C05488=1125.538,-96.139,-46.252,179.561,4.488,148.877
C05489=1125.533,-95.888,-46.261,179.560,4.493,148.878
C05490=1125.527,-95.639,-46.269,179.560,4.499,148.879
C05491=1125.522,-95.389,-46.278,179.560,4.504,148.880
C05492=1125.517,-95.139,-46.287,179.559,4.508,148.882
C05493=1125.511,-94.889,-46.296,179.559,4.513,148.883
C05494=1125.506,-94.639,-46.305,179.559,4.518,148.884
C05495=1125.500,-94.389,-46.314,179.558,4.522,148.885
C05496=1125.495,-94.140,-46.323,179.558,4.528,148.886
C05497=1125.489,-93.890,-46.332,179.557,4.532,148.888
C05498=1125.484,-93.641,-46.341,179.556,4.537,148.889
C05499=1125.478,-93.390,-46.350,179.555,4.542,148.890
C05500=1125.474,-93.141,-46.360,179.555,4.547,148.891
C05501=1125.468,-92.891,-46.369,179.554,4.551,148.893
C05502=1125.463,-92.642,-46.377,179.554,4.556,148.894
C05503=1125.457,-92.392,-46.386,179.552,4.561,148.895
C05504=1125.452,-92.142,-46.395,179.552,4.565,148.896
C05505=1125.446,-91.892,-46.404,179.551,4.570,148.897
C05506=1125.441,-91.642,-46.413,179.551,4.575,148.899
C05507=1125.436,-91.393,-46.422,179.550,4.580,148.900
C05508=1125.431,-91.143,-46.431,179.549,4.585,148.901
C05509=1125.425,-90.893,-46.441,179.548,4.589,148.902
C05510=1125.419,-90.643,-46.449,179.548,4.594,148.904
C05511=1125.414,-90.394,-46.458,179.547,4.599,148.905
C05512=1125.409,-90.144,-46.467,179.547,4.604,148.906
C05513=1125.403,-89.894,-46.477,179.546,4.609,148.907
C05514=1125.398,-89.644,-46.486,179.546,4.614,148.909
C05515=1125.393,-89.394,-46.495,179.544,4.618,148.910
C05516=1125.389,-89.179,-46.503,179.544,4.622,148.911
C05517=1125.383,-88.963,-46.511,179.543,4.627,148.912
C05518=1125.379,-88.747,-46.518,179.544,4.632,148.913
C05519=1125.374,-88.532,-46.526,179.543,4.636,148.914
C05520=1125.370,-88.316,-46.534,179.543,4.640,148.915
C05521=1125.365,-88.100,-46.542,179.542,4.644,148.916
C05522=1125.360,-87.885,-46.550,179.542,4.648,148.917
C05523=1125.356,-87.669,-46.558,179.541,4.653,148.919
C05524=1125.350,-87.419,-46.567,179.541,4.658,148.920
C05525=1125.345,-87.169,-46.576,179.540,4.662,148.921
C05526=1125.339,-86.919,-46.585,179.540,4.667,148.922
C05527=1125.335,-86.670,-46.595,179.539,4.672,148.923
C05528=1125.329,-86.420,-46.604,179.538,4.677,148.925
C05529=1125.323,-86.170,-46.613,179.538,4.682,148.926
C05530=1125.318,-85.920,-46.622,179.538,4.687,148.927
C05531=1125.313,-85.670,-46.631,179.538,4.693,148.928
C05532=1125.308,-85.421,-46.641,179.537,4.697,148.929
C05533=1125.302,-85.171,-46.650,179.537,4.702,148.931
C05534=1125.297,-84.922,-46.659,179.536,4.707,148.932
C05535=1125.291,-84.671,-46.668,179.536,4.713,148.933
C05536=1125.286,-84.422,-46.678,179.535,4.717,148.934
C05537=1125.281,-84.172,-46.687,179.535,4.722,148.935
C05538=1125.275,-83.922,-46.696,179.535,4.728,148.937
C05539=1125.270,-83.673,-46.706,179.535,4.733,148.938
C05540=1125.264,-83.423,-46.715,179.534,4.738,148.939
C05541=1125.259,-83.173,-46.724,179.534,4.743,148.940
C05542=1125.254,-82.924,-46.734,179.533,4.747,148.941
C05543=1125.248,-82.674,-46.743,179.533,4.753,148.942
C05544=1125.243,-82.424,-46.752,179.533,4.758,148.944
C05545=1125.237,-82.174,-46.763,179.532,4.763,148.945
C05546=1125.232,-81.924,-46.771,179.532,4.768,148.946
C05547=1125.227,-81.674,-46.780,179.532,4.774,148.947
C05548=1125.221,-81.425,-46.791,179.532,4.779,148.949
C05549=1125.216,-81.175,-46.799,179.532,4.784,148.950
C05550=1125.210,-80.925,-46.809,179.532,4.789,148.951
C05551=1125.205,-80.676,-46.819,179.531,4.794,148.952
C05552=1125.200,-80.425,-46.828,179.531,4.799,148.953
C05553=1125.195,-80.176,-46.838,179.531,4.805,148.954
C05554=1125.190,-79.926,-46.847,179.531,4.810,148.956
C05555=1125.184,-79.676,-46.856,179.531,4.815,148.957
C05556=1125.179,-79.426,-46.866,179.531,4.820,148.958
C05557=1125.173,-79.176,-46.876,179.530,4.825,148.959
C05558=1125.169,-78.927,-46.885,179.530,4.830,148.960
C05559=1125.163,-78.677,-46.895,179.530,4.836,148.961
C05560=1125.158,-78.427,-46.904,179.530,4.841,148.963
C05561=1125.152,-78.177,-46.914,179.530,4.846,148.964
C05562=1125.147,-77.928,-46.923,179.530,4.851,148.965
C05563=1125.141,-77.678,-46.933,179.530,4.856,148.966
C05564=1125.136,-77.429,-46.942,179.530,4.861,148.967
C05565=1125.130,-77.179,-46.952,179.530,4.867,148.968
C05566=1125.125,-76.929,-46.962,179.530,4.872,148.969
C05567=1125.120,-76.679,-46.971,179.530,4.877,148.970
C05568=1125.114,-76.430,-46.981,179.530,4.882,148.972
C05569=1125.109,-76.180,-46.990,179.530,4.888,148.973
C05570=1125.104,-75.930,-47.001,179.530,4.892,148.974
C05571=1125.099,-75.680,-47.010,179.530,4.898,148.975
C05572=1125.093,-75.465,-47.019,179.530,4.902,148.976
C05573=1125.089,-75.249,-47.027,179.530,4.907,148.977
C05574=1125.084,-75.033,-47.035,179.530,4.911,148.978
C05575=1125.080,-74.817,-47.043,179.530,4.916,148.979
C05576=1125.075,-74.602,-47.052,179.531,4.921,148.980
C05577=1125.071,-74.387,-47.060,179.530,4.925,148.981
C05578=1125.066,-74.170,-47.069,179.531,4.930,148.982
C05579=1125.062,-73.955,-47.077,179.531,4.934,148.983
C05580=1125.056,-73.705,-47.087,179.531,4.940,148.984
C05581=1125.050,-73.456,-47.097,179.531,4.945,148.985
C05582=1125.045,-73.206,-47.107,179.532,4.950,148.986
C05583=1125.039,-72.956,-47.116,179.532,4.955,148.987
C05584=1125.035,-72.706,-47.126,179.531,4.961,148.988
C05585=1125.030,-72.457,-47.136,179.532,4.966,148.989
C05586=1125.024,-72.207,-47.146,179.532,4.971,148.990
C05587=1125.019,-71.957,-47.155,179.532,4.976,148.991
C05588=1125.013,-71.708,-47.166,179.533,4.982,148.992
C05589=1125.007,-71.458,-47.175,179.533,4.987,148.993
C05590=1125.002,-71.207,-47.186,179.533,4.992,148.995
C05591=1124.997,-70.958,-47.195,179.534,4.998,148.996
C05592=1124.992,-70.709,-47.205,179.534,5.003,148.997
C05593=1124.986,-70.458,-47.215,179.535,5.009,148.998
C05594=1124.982,-70.208,-47.225,179.534,5.014,148.999
C05595=1124.976,-69.959,-47.235,179.535,5.019,149.000
C05596=1124.971,-69.709,-47.245,179.535,5.025,149.001
C05597=1124.965,-69.460,-47.256,179.536,5.029,149.002
C05598=1124.960,-69.210,-47.264,179.536,5.035,149.003
C05599=1124.955,-68.960,-47.275,179.536,5.040,149.004
C05600=1124.949,-68.710,-47.285,179.537,5.046,149.005
C05601=1124.944,-68.461,-47.295,179.537,5.051,149.006
C05602=1124.939,-68.211,-47.305,179.538,5.057,149.007
C05603=1124.934,-67.961,-47.316,179.538,5.061,149.008
C05604=1124.928,-67.711,-47.325,179.539,5.067,149.009
C05605=1124.922,-67.461,-47.335,179.539,5.072,149.010
C05606=1124.917,-67.212,-47.345,179.540,5.078,149.011
C05607=1124.912,-66.962,-47.356,179.540,5.083,149.012
C05608=1124.907,-66.712,-47.366,179.541,5.089,149.013
C05609=1124.901,-66.463,-47.376,179.541,5.093,149.014
C05610=1124.896,-66.213,-47.387,179.542,5.099,149.015
C05611=1124.891,-65.963,-47.397,179.543,5.104,149.016
C05612=1124.886,-65.714,-47.406,179.543,5.110,149.017
C05613=1124.881,-65.464,-47.417,179.543,5.114,149.018
C05614=1124.875,-65.214,-47.427,179.544,5.120,149.019
C05615=1124.869,-64.965,-47.437,179.545,5.125,149.020
C05616=1124.864,-64.714,-47.448,179.545,5.131,149.021
C05617=1124.859,-64.465,-47.458,179.546,5.136,149.022
C05618=1124.853,-64.215,-47.468,179.547,5.141,149.023
C05619=1124.848,-63.965,-47.479,179.548,5.147,149.024
C05620=1124.843,-63.716,-47.489,179.549,5.152,149.024
C05621=1124.838,-63.466,-47.499,179.549,5.157,149.025
C05622=1124.833,-63.216,-47.509,179.550,5.162,149.026
C05623=1124.827,-62.966,-47.519,179.551,5.168,149.027
C05624=1124.822,-62.717,-47.530,179.551,5.173,149.028
C05625=1124.817,-62.467,-47.540,179.552,5.178,149.029
C05626=1124.811,-62.218,-47.551,179.553,5.184,149.030
C05627=1124.806,-61.967,-47.562,179.554,5.189,149.031
C05628=1124.801,-61.751,-47.570,179.554,5.193,149.032
C05629=1124.797,-61.536,-47.580,179.555,5.198,149.032
C05630=1124.793,-61.321,-47.588,179.556,5.203,149.033
C05631=1124.788,-61.106,-47.597,179.557,5.208,149.034
C05632=1124.783,-60.890,-47.607,179.558,5.212,149.035
C05633=1124.778,-60.675,-47.616,179.559,5.216,149.035
C05634=1124.773,-60.459,-47.624,179.559,5.221,149.036
C05635=1124.769,-60.244,-47.633,179.560,5.226,149.037
C05636=1124.765,-59.994,-47.644,179.559,5.230,149.038
C05637=1124.759,-59.744,-47.655,179.560,5.235,149.039
C05638=1124.754,-59.494,-47.665,179.559,5.240,149.040
C05639=1124.749,-59.245,-47.675,179.559,5.244,149.041
C05640=1124.743,-58.994,-47.687,179.559,5.249,149.042
C05641=1124.738,-58.745,-47.697,179.558,5.253,149.043
C05642=1124.733,-58.495,-47.708,179.559,5.258,149.044
C05643=1124.727,-58.245,-47.718,179.558,5.262,149.046
C05644=1124.722,-57.996,-47.730,179.558,5.268,149.047
C05645=1124.717,-57.746,-47.740,179.558,5.271,149.048
C05646=1124.712,-57.496,-47.750,179.558,5.277,149.049
C05647=1124.706,-57.246,-47.761,179.557,5.281,149.050
C05648=1124.701,-56.997,-47.772,179.557,5.286,149.051
C05649=1124.696,-56.747,-47.782,179.557,5.291,149.052
C05650=1124.691,-56.497,-47.793,179.557,5.295,149.053
C05651=1124.685,-56.248,-47.804,179.557,5.300,149.054
C05652=1124.680,-55.998,-47.814,179.556,5.304,149.055
C05653=1124.675,-55.748,-47.824,179.556,5.309,149.056
C05654=1124.669,-55.498,-47.836,179.556,5.313,149.057
C05655=1124.664,-55.249,-47.846,179.556,5.319,149.058
C05656=1124.659,-54.999,-47.857,179.556,5.324,149.060
C05657=1124.654,-54.750,-47.868,179.556,5.328,149.060
C05658=1124.649,-54.499,-47.879,179.556,5.333,149.062
C05659=1124.643,-54.250,-47.889,179.555,5.337,149.063
C05660=1124.638,-54.000,-47.900,179.555,5.342,149.064
C05661=1124.632,-53.750,-47.911,179.555,5.346,149.065
C05662=1124.627,-53.501,-47.922,179.555,5.351,149.066
C05663=1124.622,-53.251,-47.932,179.554,5.355,149.067
C05664=1124.617,-53.002,-47.944,179.554,5.361,149.068
C05665=1124.611,-52.752,-47.954,179.554,5.366,149.069
C05666=1124.607,-52.502,-47.965,179.554,5.370,149.070
C05667=1124.600,-52.253,-47.976,179.554,5.375,149.071
C05668=1124.595,-52.002,-47.986,179.553,5.379,149.072
C05669=1124.590,-51.753,-47.997,179.553,5.384,149.074
C05670=1124.585,-51.503,-48.008,179.553,5.388,149.074
C05671=1124.580,-51.254,-48.019,179.553,5.393,149.076
C05672=1124.574,-51.004,-48.030,179.553,5.398,149.077
C05673=1124.569,-50.754,-48.041,179.553,5.402,149.078
C05674=1124.564,-50.504,-48.052,179.553,5.408,149.079
C05675=1124.559,-50.255,-48.063,179.552,5.412,149.080
C05676=1124.553,-50.005,-48.074,179.552,5.417,149.081
C05677=1124.548,-49.755,-48.085,179.552,5.421,149.082
C05678=1124.543,-49.505,-48.096,179.552,5.426,149.083
C05679=1124.538,-49.256,-48.106,179.551,5.431,149.084
C05680=1124.532,-49.006,-48.118,179.551,5.435,149.085
C05681=1124.527,-48.757,-48.129,179.551,5.440,149.086
C05682=1124.522,-48.507,-48.140,179.551,5.445,149.088
C05683=1124.517,-48.257,-48.150,179.551,5.450,149.088
C05684=1124.512,-48.041,-48.160,179.551,5.453,149.089
C05685=1124.508,-47.827,-48.170,179.550,5.458,149.090
C05686=1124.503,-47.611,-48.179,179.550,5.462,149.091
C05687=1124.498,-47.395,-48.189,179.550,5.466,149.092
C05688=1124.493,-47.180,-48.198,179.550,5.470,149.093
C05689=1124.489,-46.964,-48.207,179.550,5.474,149.094
C05690=1124.484,-46.749,-48.217,179.550,5.478,149.095
C05691=1124.480,-46.534,-48.227,179.550,5.482,149.096
C05692=1124.475,-46.284,-48.238,179.549,5.487,149.097
C05693=1124.470,-46.034,-48.249,179.549,5.491,149.098
C05694=1124.464,-45.785,-48.260,179.549,5.496,149.099
C05695=1124.459,-45.535,-48.271,179.549,5.501,149.100
C05696=1124.454,-45.285,-48.282,179.549,5.506,149.101
C05697=1124.448,-45.036,-48.294,179.548,5.510,149.102
C05698=1124.443,-44.785,-48.304,179.548,5.515,149.103
C05699=1124.439,-44.536,-48.315,179.548,5.519,149.105
C05700=1124.433,-44.287,-48.327,179.548,5.525,149.106
C05701=1124.428,-44.037,-48.338,179.548,5.529,149.107
C05702=1124.423,-43.787,-48.349,179.547,5.534,149.108
C05703=1124.417,-43.537,-48.360,179.547,5.539,149.109
C05704=1124.412,-43.288,-48.372,179.547,5.543,149.110
C05705=1124.406,-43.037,-48.383,179.548,5.549,149.111
C05706=1124.401,-42.788,-48.394,179.549,5.554,149.112
C05707=1124.396,-42.539,-48.405,179.551,5.560,149.112
C05708=1124.391,-42.289,-48.417,179.552,5.565,149.113
C05709=1124.385,-42.039,-48.427,179.555,5.571,149.114
C05710=1124.380,-41.789,-48.439,179.556,5.577,149.115
C05711=1124.375,-41.540,-48.450,179.558,5.583,149.115
C05712=1124.370,-41.290,-48.462,179.559,5.588,149.116
C05713=1124.365,-41.041,-48.473,179.561,5.594,149.117
C05714=1124.359,-40.791,-48.485,179.563,5.599,149.117
C05715=1124.354,-40.541,-48.495,179.564,5.605,149.118
C05716=1124.349,-40.291,-48.507,179.566,5.610,149.119
C05717=1124.343,-40.042,-48.518,179.567,5.615,149.120
C05718=1124.338,-39.792,-48.530,179.568,5.621,149.121
C05719=1124.333,-39.542,-48.541,179.570,5.626,149.121
C05720=1124.328,-39.292,-48.553,179.571,5.631,149.122
C05721=1124.323,-39.043,-48.564,179.572,5.636,149.123
C05722=1124.317,-38.793,-48.576,179.574,5.642,149.123
C05723=1124.312,-38.544,-48.587,179.575,5.647,149.124
C05724=1124.307,-38.294,-48.599,179.576,5.651,149.125
C05725=1124.302,-38.044,-48.611,179.577,5.657,149.126
C05726=1124.296,-37.795,-48.622,179.578,5.661,149.127
C05727=1124.291,-37.545,-48.634,179.579,5.667,149.127
C05728=1124.286,-37.295,-48.645,179.580,5.672,149.128
C05729=1124.281,-37.045,-48.657,179.581,5.676,149.129
C05730=1124.275,-36.796,-48.669,179.582,5.681,149.130
C05731=1124.271,-36.546,-48.680,179.583,5.686,149.130
C05732=1124.265,-36.297,-48.692,179.584,5.691,149.131
C05733=1124.260,-36.047,-48.703,179.585,5.695,149.132
C05734=1124.254,-35.797,-48.715,179.585,5.700,149.133
C05735=1124.249,-35.547,-48.727,179.586,5.706,149.134
C05736=1124.244,-35.298,-48.738,179.587,5.710,149.134
C05737=1124.239,-35.048,-48.750,179.588,5.715,149.135
C05738=1124.234,-34.798,-48.763,179.588,5.720,149.136
C05739=1124.229,-34.549,-48.774,179.589,5.724,149.137
C05740=1124.224,-34.333,-48.785,179.589,5.728,149.138
C05741=1124.219,-34.118,-48.794,179.589,5.731,149.138
C05742=1124.215,-33.903,-48.804,179.590,5.736,149.139
C05743=1124.211,-33.687,-48.815,179.590,5.739,149.140
C05744=1124.206,-33.472,-48.825,179.590,5.743,149.141
C05745=1124.201,-33.257,-48.835,179.591,5.747,149.141
C05746=1124.197,-33.041,-48.845,179.591,5.750,149.142
C05747=1124.193,-32.826,-48.855,179.591,5.755,149.143
C05748=1124.187,-32.576,-48.867,179.591,5.759,149.144
C05749=1124.182,-32.326,-48.879,179.592,5.764,149.145
C05750=1124.177,-32.077,-48.892,179.592,5.768,149.146
C05751=1124.172,-31.827,-48.903,179.592,5.773,149.147
C05752=1124.167,-31.577,-48.915,179.592,5.776,149.147
C05753=1124.161,-31.327,-48.927,179.592,5.780,149.148
C05754=1124.156,-31.078,-48.939,179.592,5.785,149.149
C05755=1124.151,-30.828,-48.950,179.592,5.789,149.150
C05756=1124.145,-30.579,-48.962,179.591,5.793,149.151
C05757=1124.140,-30.329,-48.974,179.591,5.797,149.152
C05758=1124.135,-30.080,-48.986,179.592,5.802,149.153
C05759=1124.130,-29.830,-48.998,179.592,5.806,149.154
C05760=1124.125,-29.580,-49.010,179.591,5.810,149.155
C05761=1124.120,-29.331,-49.022,179.591,5.814,149.156
C05762=1124.114,-29.081,-49.034,179.590,5.819,149.157
C05763=1124.109,-28.831,-49.046,179.590,5.823,149.158
C05764=1124.104,-28.582,-49.057,179.589,5.826,149.159
C05765=1124.099,-28.332,-49.070,179.588,5.831,149.160
C05766=1124.093,-28.082,-49.082,179.588,5.834,149.161
C05767=1124.088,-27.832,-49.094,179.587,5.839,149.162
C05768=1124.083,-27.583,-49.106,179.587,5.843,149.164
C05769=1124.078,-27.333,-49.118,179.586,5.847,149.165
C05770=1124.073,-27.084,-49.129,179.585,5.851,149.166
C05771=1124.068,-26.834,-49.142,179.585,5.855,149.167
C05772=1124.062,-26.584,-49.154,179.584,5.858,149.168
C05773=1124.057,-26.335,-49.167,179.583,5.863,149.169
C05774=1124.052,-26.085,-49.178,179.581,5.867,149.170
C05775=1124.047,-25.835,-49.190,179.582,5.871,149.171
C05776=1124.042,-25.586,-49.202,179.582,5.876,149.172
C05777=1124.036,-25.336,-49.214,179.583,5.881,149.173
C05778=1124.031,-25.086,-49.226,179.584,5.886,149.174
C05779=1124.026,-24.837,-49.239,179.584,5.891,149.175
C05780=1124.020,-24.587,-49.251,179.585,5.896,149.175
C05781=1124.015,-24.338,-49.263,179.586,5.901,149.176
C05782=1124.010,-24.088,-49.275,179.587,5.906,149.177
C05783=1124.006,-23.839,-49.287,179.587,5.911,149.178
C05784=1124.000,-23.589,-49.299,179.588,5.915,149.179
C05785=1123.995,-23.339,-49.312,179.589,5.921,149.180
C05786=1123.990,-23.090,-49.323,179.590,5.925,149.181
C05787=1123.984,-22.840,-49.336,179.590,5.930,149.182
C05788=1123.979,-22.590,-49.348,179.591,5.935,149.182
C05789=1123.974,-22.341,-49.361,179.592,5.940,149.183
C05790=1123.969,-22.090,-49.373,179.592,5.945,149.184
C05791=1123.964,-21.841,-49.385,179.593,5.950,149.185
C05792=1123.958,-21.591,-49.397,179.594,5.954,149.186
C05793=1123.953,-21.342,-49.410,179.595,5.960,149.187
C05794=1123.948,-21.092,-49.422,179.595,5.964,149.188
C05795=1123.943,-20.842,-49.434,179.596,5.969,149.188
C05796=1123.938,-20.627,-49.445,179.597,5.973,149.189
C05797=1123.934,-20.412,-49.455,179.597,5.977,149.190
C05798=1123.929,-20.197,-49.466,179.598,5.981,149.190
C05799=1123.925,-19.982,-49.477,179.598,5.985,149.191
C05800=1123.920,-19.766,-49.488,179.599,5.990,149.192
C05801=1123.916,-19.551,-49.499,179.600,5.994,149.193
C05802=1123.912,-19.336,-49.509,179.600,5.997,149.193
C05803=1123.907,-19.120,-49.520,179.601,6.002,149.194
C05804=1123.902,-18.870,-49.532,179.602,6.007,149.195
C05805=1123.897,-18.621,-49.545,179.602,6.011,149.196
C05806=1123.891,-18.371,-49.557,179.603,6.016,149.197
C05807=1123.886,-18.122,-49.569,179.603,6.021,149.198
C05808=1123.881,-17.873,-49.582,179.605,6.026,149.198
C05809=1123.876,-17.623,-49.594,179.605,6.031,149.199
C05810=1123.870,-17.372,-49.607,179.606,6.035,149.200
C05811=1123.865,-17.123,-49.620,179.607,6.040,149.201
C05812=1123.860,-16.874,-49.633,179.607,6.044,149.202
C05813=1123.855,-16.624,-49.644,179.608,6.049,149.202
C05814=1123.850,-16.374,-49.657,179.608,6.054,149.203
C05815=1123.845,-16.125,-49.670,179.609,6.058,149.204
C05816=1123.840,-15.875,-49.683,179.610,6.064,149.205
C05817=1123.835,-15.625,-49.694,179.611,6.069,149.206
C05818=1123.829,-15.376,-49.707,179.612,6.073,149.206
C05819=1123.824,-15.126,-49.720,179.612,6.078,149.207
C05820=1123.818,-14.877,-49.733,179.613,6.082,149.208
C05821=1123.814,-14.627,-49.746,179.614,6.087,149.209
C05822=1123.809,-14.378,-49.758,179.614,6.091,149.210
C05823=1123.803,-14.128,-49.770,179.615,6.096,149.211
C05824=1123.798,-13.878,-49.783,179.615,6.101,149.212
C05825=1123.793,-13.628,-49.796,179.616,6.105,149.212
C05826=1123.788,-13.379,-49.809,179.617,6.110,149.213
C05827=1123.783,-13.129,-49.822,179.617,6.115,149.214
C05828=1123.778,-12.880,-49.834,179.618,6.119,149.215
C05829=1123.773,-12.630,-49.847,179.619,6.124,149.216
C05830=1123.767,-12.380,-49.860,179.619,6.128,149.216
C05831=1123.762,-12.131,-49.873,179.620,6.133,149.217
C05832=1123.757,-11.882,-49.886,179.621,6.138,149.218
C05833=1123.752,-11.631,-49.898,179.621,6.142,149.219
C05834=1123.746,-11.381,-49.911,179.622,6.147,149.220
C05835=1123.741,-11.132,-49.924,179.623,6.151,149.220
C05836=1123.737,-10.882,-49.937,179.623,6.156,149.221
C05837=1123.732,-10.633,-49.949,179.624,6.160,149.222
C05838=1123.726,-10.383,-49.962,179.625,6.165,149.223
C05839=1123.721,-10.134,-49.975,179.625,6.170,149.224
C05840=1123.716,-9.884,-49.988,179.626,6.174,149.224
C05841=1123.710,-9.634,-50.001,179.627,6.179,149.225
C05842=1123.705,-9.385,-50.014,179.627,6.184,149.226
C05843=1123.701,-9.135,-50.027,179.628,6.188,149.227
C05844=1123.695,-8.886,-50.041,179.629,6.193,149.228
C05845=1123.690,-8.637,-50.053,179.629,6.197,149.229
C05846=1123.685,-8.387,-50.066,179.630,6.202,149.229
C05847=1123.679,-8.137,-50.079,179.631,6.207,149.230
C05848=1123.674,-7.888,-50.092,179.631,6.211,149.231
C05849=1123.670,-7.638,-50.105,179.632,6.216,149.232
C05850=1123.664,-7.388,-50.118,179.633,6.220,149.233
C05851=1123.659,-7.139,-50.131,179.633,6.225,149.233
C05852=1123.655,-6.923,-50.142,179.634,6.229,149.234
C05853=1123.651,-6.708,-50.154,179.635,6.233,149.235
C05854=1123.645,-6.493,-50.165,179.635,6.236,149.235
C05855=1123.641,-6.278,-50.176,179.636,6.241,149.236
C05856=1123.637,-6.062,-50.188,179.636,6.245,149.237
C05857=1123.632,-5.847,-50.199,179.636,6.248,149.238
C05858=1123.628,-5.632,-50.210,179.637,6.253,149.238
C05859=1123.624,-5.417,-50.221,179.638,6.256,149.239
C05860=1123.619,-5.167,-50.235,179.638,6.261,149.240
C05861=1123.613,-4.918,-50.247,179.639,6.265,149.241
C05862=1123.608,-4.668,-50.261,179.640,6.270,149.241
C05863=1123.603,-4.419,-50.274,179.640,6.275,149.242
C05864=1123.598,-4.169,-50.288,179.641,6.279,149.243
C05865=1123.593,-3.919,-50.300,179.641,6.283,149.244
C05866=1123.587,-3.670,-50.314,179.642,6.288,149.245
C05867=1123.583,-3.420,-50.327,179.642,6.292,149.246
C05868=1123.577,-3.171,-50.340,179.643,6.297,149.246
C05869=1123.572,-2.921,-50.353,179.644,6.301,149.247
C05870=1123.567,-2.671,-50.367,179.644,6.306,149.248
C05871=1123.562,-2.422,-50.380,179.645,6.311,149.249
C05872=1123.557,-2.172,-50.393,179.646,6.315,149.250
C05873=1123.551,-1.923,-50.406,179.646,6.320,149.250
C05874=1123.546,-1.673,-50.420,179.646,6.324,149.251
C05875=1123.541,-1.424,-50.433,179.647,6.328,149.252
C05876=1123.536,-1.173,-50.446,179.648,6.333,149.253
C05877=1123.531,-0.925,-50.460,179.648,6.338,149.254
C05878=1123.526,-0.674,-50.473,179.649,6.342,149.255
C05879=1123.521,-0.425,-50.486,179.650,6.347,149.255
C05880=1123.516,-0.175,-50.500,179.650,6.351,149.256
C05881=1123.511,0.074,-50.513,179.650,6.355,149.257
C05882=1123.506,0.324,-50.527,179.651,6.360,149.258
C05883=1123.500,0.573,-50.540,179.652,6.364,149.259
C05884=1123.495,0.823,-50.553,179.652,6.369,149.260
C05885=1123.490,1.072,-50.567,179.653,6.374,149.260
C05886=1123.485,1.322,-50.580,179.653,6.379,149.261
C05887=1123.480,1.571,-50.594,179.654,6.382,149.262
C05888=1123.475,1.821,-50.607,179.654,6.387,149.263
C05889=1123.470,2.070,-50.621,179.655,6.392,149.264
C05890=1123.464,2.321,-50.635,179.655,6.396,149.265
C05891=1123.460,2.569,-50.648,179.656,6.401,149.265
C05892=1123.454,2.820,-50.661,179.657,6.405,149.266
C05893=1123.449,3.069,-50.675,179.657,6.409,149.267
C05894=1123.444,3.319,-50.688,179.657,6.414,149.268
C05895=1123.439,3.568,-50.702,179.658,6.419,149.269
C05896=1123.434,3.818,-50.716,179.658,6.423,149.270
C05897=1123.429,4.068,-50.729,179.659,6.428,149.270
C05898=1123.423,4.317,-50.743,179.660,6.432,149.271
C05899=1123.418,4.567,-50.757,179.660,6.436,149.272
C05900=1123.413,4.816,-50.769,179.660,6.441,149.273
C05901=1123.408,5.066,-50.784,179.661,6.446,149.274
C05902=1123.403,5.315,-50.798,179.661,6.451,149.275
C05903=1123.398,5.565,-50.811,179.662,6.455,149.275
C05904=1123.393,5.815,-50.825,179.662,6.459,149.276
C05905=1123.388,6.064,-50.838,179.663,6.464,149.277
C05906=1123.383,6.314,-50.852,179.664,6.468,149.278
C05907=1123.378,6.563,-50.866,179.664,6.473,149.279
C05908=1123.374,6.778,-50.877,179.664,6.477,149.280
C05909=1123.369,6.994,-50.890,179.664,6.480,149.280
C05910=1123.364,7.209,-50.901,179.665,6.485,149.281
C05911=1123.360,7.423,-50.913,179.666,6.488,149.282
C05912=1123.356,7.639,-50.924,179.666,6.492,149.283
C05913=1123.351,7.854,-50.937,179.666,6.496,149.283
C05914=1123.347,8.069,-50.949,179.667,6.501,149.284
C05915=1123.343,8.284,-50.961,179.667,6.504,149.285
C05916=1123.337,8.533,-50.975,179.668,6.509,149.286
C05917=1123.332,8.783,-50.988,179.669,6.513,149.286
C05918=1123.328,9.033,-51.002,179.669,6.518,149.287
C05919=1123.322,9.282,-51.016,179.670,6.523,149.288
C05920=1123.317,9.532,-51.030,179.671,6.528,149.289
C05921=1123.312,9.782,-51.044,179.672,6.532,149.290
C05922=1123.306,10.031,-51.058,179.673,6.537,149.291
C05923=1123.302,10.280,-51.071,179.674,6.541,149.291
C05924=1123.297,10.530,-51.085,179.674,6.546,149.292
C05925=1123.292,10.779,-51.099,179.675,6.551,149.293
C05926=1123.286,11.029,-51.113,179.676,6.555,149.294
C05927=1123.281,11.279,-51.127,179.676,6.560,149.295
C05928=1123.276,11.528,-51.141,179.678,6.565,149.295
C05929=1123.271,11.778,-51.155,179.678,6.570,149.296
C05930=1123.267,12.027,-51.169,179.679,6.574,149.297
C05931=1123.261,12.277,-51.182,179.680,6.579,149.298
C05932=1123.256,12.527,-51.197,179.681,6.583,149.298
C05933=1123.251,12.776,-51.211,179.682,6.588,149.299
C05934=1123.246,13.026,-51.225,179.682,6.592,149.300
C05935=1123.240,13.275,-51.239,179.683,6.597,149.301
C05936=1123.235,13.525,-51.253,179.684,6.602,149.302
C05937=1123.230,13.774,-51.268,179.685,6.606,149.302
C05938=1123.225,14.023,-51.282,179.686,6.611,149.303
C05939=1123.220,14.273,-51.296,179.687,6.616,149.304
C05940=1123.215,14.523,-51.310,179.687,6.620,149.305
C05941=1123.210,14.773,-51.324,179.689,6.625,149.305
C05942=1123.204,15.022,-51.338,179.689,6.629,149.306
C05943=1123.199,15.271,-51.353,179.690,6.634,149.307
C05944=1123.195,15.521,-51.367,179.691,6.638,149.308
C05945=1123.190,15.771,-51.381,179.692,6.643,149.308
C05946=1123.185,16.020,-51.395,179.692,6.647,149.309
C05947=1123.179,16.269,-51.409,179.693,6.652,149.310
C05948=1123.174,16.519,-51.424,179.694,6.657,149.311
C05949=1123.169,16.769,-51.438,179.695,6.661,149.311
C05950=1123.164,17.019,-51.452,179.697,6.666,149.312
C05951=1123.159,17.268,-51.466,179.697,6.671,149.313
C05952=1123.154,17.517,-51.480,179.698,6.675,149.314
C05953=1123.149,17.767,-51.495,179.699,6.680,149.314
C05954=1123.144,18.017,-51.509,179.700,6.684,149.315
C05955=1123.139,18.266,-51.523,179.701,6.688,149.316
C05956=1123.134,18.516,-51.537,179.701,6.693,149.317
C05957=1123.128,18.765,-51.551,179.702,6.697,149.317
C05958=1123.124,19.014,-51.566,179.703,6.702,149.318
C05959=1123.119,19.264,-51.581,179.704,6.706,149.319
C05960=1123.114,19.514,-51.595,179.705,6.711,149.319
C05961=1123.109,19.763,-51.609,179.706,6.715,149.320
C05962=1123.104,20.013,-51.623,179.707,6.720,149.321
C05963=1123.098,20.262,-51.638,179.708,6.724,149.322
C05964=1123.094,20.477,-51.650,179.709,6.728,149.322
C05965=1123.089,20.692,-51.663,179.709,6.732,149.323
C05966=1123.085,20.907,-51.675,179.710,6.736,149.324
C05967=1123.080,21.122,-51.688,179.711,6.739,149.324
C05968=1123.076,21.337,-51.700,179.712,6.744,149.325
C05969=1123.072,21.552,-51.713,179.713,6.747,149.325
C05970=1123.068,21.767,-51.725,179.714,6.752,149.326
C05971=1123.063,21.982,-51.738,179.714,6.755,149.327
C05972=1123.058,22.232,-51.752,179.715,6.759,149.327
C05973=1123.053,22.481,-51.767,179.716,6.764,149.328
C05974=1123.048,22.730,-51.782,179.717,6.768,149.329
C05975=1123.043,22.981,-51.796,179.718,6.773,149.329
C05976=1123.038,23.230,-51.811,179.719,6.777,149.330
C05977=1123.033,23.479,-51.826,179.720,6.781,149.331
C05978=1123.028,23.729,-51.840,179.721,6.786,149.331
C05979=1123.023,23.979,-51.854,179.722,6.790,149.332
C05980=1123.018,24.228,-51.870,179.723,6.795,149.333
C05981=1123.013,24.478,-51.884,179.724,6.799,149.334
C05982=1123.008,24.728,-51.898,179.725,6.804,149.334
C05983=1123.003,24.976,-51.913,179.726,6.808,149.335
C05984=1122.997,25.226,-51.928,179.727,6.813,149.336
C05985=1122.992,25.475,-51.943,179.728,6.818,149.336
C05986=1122.987,25.725,-51.957,179.729,6.822,149.337
C05987=1122.982,25.974,-51.971,179.730,6.826,149.338
C05988=1122.977,26.224,-51.987,179.731,6.830,149.338
C05989=1122.972,26.474,-52.001,179.732,6.835,149.339
C05990=1122.967,26.723,-52.016,179.733,6.839,149.340
C05991=1122.962,26.973,-52.031,179.734,6.843,149.340
C05992=1122.957,27.222,-52.046,179.735,6.848,149.341
C05993=1122.952,27.471,-52.060,179.736,6.852,149.342
C05994=1122.947,27.721,-52.076,179.737,6.857,149.342
C05995=1122.942,27.971,-52.090,179.738,6.861,149.343
C05996=1122.937,28.220,-52.105,179.739,6.865,149.344
C05997=1122.932,28.470,-52.120,179.740,6.870,149.344
C05998=1122.927,28.719,-52.135,179.741,6.874,149.345
C05999=1122.922,28.969,-52.149,179.742,6.878,149.346
C06000=1122.917,29.218,-52.165,179.743,6.883,149.346
C06001=1122.912,29.468,-52.179,179.744,6.887,149.347
C06002=1122.906,29.717,-52.195,179.745,6.891,149.348
C06003=1122.902,29.966,-52.210,179.746,6.896,149.348
C06004=1122.897,30.217,-52.225,179.748,6.900,149.349
C06005=1122.892,30.466,-52.240,179.749,6.904,149.350
C06006=1122.887,30.716,-52.254,179.750,6.909,149.350
C06007=1122.881,30.965,-52.270,179.751,6.913,149.351
C06008=1122.877,31.214,-52.285,179.752,6.917,149.352
C06009=1122.871,31.464,-52.300,179.753,6.921,149.352
C06010=1122.866,31.713,-52.315,179.754,6.926,149.353
C06011=1122.862,31.962,-52.330,179.755,6.930,149.354
C06012=1122.856,32.212,-52.345,179.756,6.934,149.354
C06013=1122.851,32.461,-52.360,179.757,6.939,149.355
C06014=1122.846,32.711,-52.375,179.758,6.943,149.355
C06015=1122.841,32.961,-52.390,179.759,6.947,149.356
C06016=1122.836,33.211,-52.406,179.760,6.951,149.357
C06017=1122.832,33.460,-52.421,179.761,6.955,149.357
C06018=1122.826,33.709,-52.436,179.762,6.959,149.358
C06019=1122.821,33.959,-52.450,179.763,6.964,149.359
C06020=1122.817,34.173,-52.464,179.764,6.968,149.359
C06021=1122.812,34.388,-52.477,179.765,6.971,149.360
C06022=1122.808,34.603,-52.490,179.766,6.975,149.360
C06023=1122.804,34.819,-52.503,179.767,6.979,149.361
C06024=1122.799,35.034,-52.516,179.768,6.983,149.361
C06025=1122.796,35.248,-52.530,179.769,6.986,149.362
C06026=1122.791,35.463,-52.543,179.770,6.989,149.362
C06027=1122.786,35.678,-52.556,179.771,6.993,149.363
C06028=1122.781,35.927,-52.571,179.772,6.997,149.363
C06029=1122.777,36.177,-52.587,179.773,7.002,149.364
C06030=1122.772,36.426,-52.602,179.774,7.006,149.365
C06031=1122.766,36.676,-52.617,179.775,7.010,149.365
C06032=1122.761,36.925,-52.632,179.777,7.015,149.366
C06033=1122.756,37.175,-52.648,179.778,7.019,149.367
C06034=1122.751,37.424,-52.663,179.779,7.023,149.367
C06035=1122.746,37.674,-52.678,179.780,7.027,149.368
C06036=1122.741,37.923,-52.694,179.781,7.031,149.368
C06037=1122.736,38.172,-52.709,179.782,7.035,149.369
C06038=1122.731,38.422,-52.725,179.783,7.039,149.370
C06039=1122.726,38.671,-52.740,179.784,7.044,149.370
C06040=1122.722,38.921,-52.756,179.785,7.048,149.371
C06041=1122.716,39.170,-52.771,179.786,7.052,149.371
C06042=1122.711,39.420,-52.787,179.788,7.056,149.372
C06043=1122.706,39.669,-52.802,179.789,7.061,149.373
C06044=1122.701,39.919,-52.818,179.790,7.064,149.373
C06045=1122.696,40.168,-52.833,179.791,7.069,149.374
C06046=1122.691,40.418,-52.848,179.792,7.073,149.374
C06047=1122.686,40.667,-52.864,179.793,7.077,149.375
C06048=1122.681,40.917,-52.880,179.795,7.081,149.376
C06049=1122.676,41.166,-52.895,179.796,7.086,149.376
C06050=1122.671,41.416,-52.910,179.797,7.090,149.377
C06051=1122.666,41.665,-52.926,179.798,7.094,149.377
C06052=1122.661,41.915,-52.942,179.800,7.098,149.378
C06053=1122.656,42.164,-52.958,179.801,7.102,149.379
C06054=1122.651,42.414,-52.973,179.802,7.107,149.379
C06055=1122.646,42.664,-52.989,179.803,7.111,149.380
C06056=1122.641,42.912,-53.005,179.804,7.115,149.380
C06057=1122.636,43.162,-53.020,179.806,7.119,149.381
C06058=1122.631,43.411,-53.035,179.806,7.123,149.382
C06059=1122.626,43.661,-53.051,179.808,7.127,149.382
C06060=1122.621,43.910,-53.067,179.809,7.131,149.383
C06061=1122.616,44.160,-53.083,179.810,7.135,149.383
C06062=1122.611,44.409,-53.099,179.811,7.139,149.384
C06063=1122.606,44.658,-53.114,179.812,7.144,149.384
C06064=1122.601,44.908,-53.130,179.813,7.148,149.385
C06065=1122.596,45.158,-53.146,179.815,7.152,149.385
C06066=1122.591,45.407,-53.161,179.816,7.156,149.386
C06067=1122.586,45.656,-53.178,179.817,7.160,149.387
C06068=1122.581,45.906,-53.194,179.819,7.164,149.387
C06069=1122.576,46.156,-53.209,179.820,7.169,149.388
C06070=1122.572,46.405,-53.225,179.821,7.173,149.388
C06071=1122.566,46.654,-53.241,179.822,7.177,149.389
C06072=1122.561,46.904,-53.256,179.823,7.181,149.390
C06073=1122.556,47.154,-53.272,179.825,7.185,149.390
C06074=1122.551,47.402,-53.289,179.826,7.189,149.391
C06075=1122.546,47.652,-53.304,179.827,7.193,149.391
C06076=1122.542,47.867,-53.318,179.828,7.197,149.392
C06077=1122.538,48.081,-53.332,179.829,7.200,149.392
C06078=1122.534,48.297,-53.345,179.831,7.204,149.393
C06079=1122.529,48.512,-53.360,179.831,7.207,149.393
C06080=1122.524,48.726,-53.373,179.832,7.210,149.394
C06081=1122.520,48.942,-53.387,179.834,7.214,149.394
C06082=1122.516,49.156,-53.400,179.834,7.218,149.395
C06083=1122.512,49.370,-53.414,179.836,7.222,149.395
C06084=1122.507,49.620,-53.430,179.836,7.225,149.396
C06085=1122.502,49.869,-53.446,179.838,7.229,149.396
C06086=1122.497,50.119,-53.462,179.839,7.233,149.397
C06087=1122.492,50.368,-53.479,179.840,7.237,149.397
C06088=1122.487,50.618,-53.495,179.842,7.241,149.398
C06089=1122.482,50.867,-53.511,179.843,7.246,149.398
C06090=1122.477,51.117,-53.527,179.844,7.250,149.399
C06091=1122.472,51.366,-53.543,179.845,7.254,149.399
C06092=1122.468,51.616,-53.559,179.847,7.258,149.400
C06093=1122.463,51.865,-53.575,179.848,7.262,149.401
C06094=1122.457,52.114,-53.591,179.849,7.266,149.401
C06095=1122.453,52.364,-53.608,179.851,7.270,149.402
C06096=1122.447,52.613,-53.623,179.852,7.275,149.402
C06097=1122.442,52.863,-53.641,179.853,7.279,149.403
C06098=1122.437,53.112,-53.656,179.855,7.283,149.403
C06099=1122.432,53.362,-53.673,179.855,7.286,149.404
C06100=1122.427,53.610,-53.689,179.857,7.290,149.404
C06101=1122.422,53.860,-53.705,179.858,7.294,149.405
C06102=1122.417,54.109,-53.721,179.859,7.298,149.405
C06103=1122.412,54.359,-53.737,179.861,7.302,149.406
C06104=1122.407,54.608,-53.754,179.862,7.307,149.407
C06105=1122.403,54.858,-53.770,179.863,7.311,149.407
C06106=1122.397,55.108,-53.787,179.864,7.315,149.408
C06107=1122.392,55.357,-53.803,179.866,7.319,149.408
C06108=1122.388,55.606,-53.820,179.867,7.323,149.409
C06109=1122.382,55.856,-53.835,179.869,7.327,149.409
C06110=1122.378,56.105,-53.852,179.870,7.331,149.410
C06111=1122.373,56.354,-53.868,179.871,7.335,149.410
C06112=1122.368,56.604,-53.884,179.872,7.340,149.411
C06113=1122.362,56.853,-53.901,179.873,7.343,149.411
C06114=1122.358,57.103,-53.918,179.875,7.347,149.412
C06115=1122.353,57.352,-53.935,179.876,7.351,149.412
C06116=1122.348,57.602,-53.950,179.878,7.355,149.413
C06117=1122.343,57.851,-53.967,179.879,7.359,149.413
C06118=1122.338,58.100,-53.984,179.880,7.363,149.414
C06119=1122.333,58.350,-54.000,179.881,7.367,149.415
C06120=1122.328,58.600,-54.016,179.883,7.371,149.415
C06121=1122.323,58.849,-54.033,179.884,7.375,149.415
C06122=1122.318,59.098,-54.050,179.886,7.379,149.416
C06123=1122.313,59.347,-54.066,179.887,7.383,149.416
C06124=1122.309,59.597,-54.083,179.888,7.388,149.417
C06125=1122.304,59.846,-54.100,179.890,7.392,149.418
C06126=1122.298,60.095,-54.116,179.891,7.395,149.418
C06127=1122.293,60.345,-54.132,179.892,7.399,149.419
C06128=1122.289,60.595,-54.149,179.893,7.403,149.419
C06129=1122.283,60.844,-54.166,179.895,7.407,149.420
C06130=1122.279,61.093,-54.183,179.896,7.411,149.420
C06131=1122.274,61.343,-54.199,179.898,7.415,149.421
C06132=1122.269,61.557,-54.214,179.899,7.419,149.421
C06133=1122.266,61.772,-54.228,179.900,7.422,149.422
C06134=1122.261,61.986,-54.243,179.901,7.425,149.422
C06135=1122.257,62.202,-54.257,179.902,7.429,149.422
C06136=1122.252,62.416,-54.271,179.903,7.433,149.423
C06137=1122.249,62.631,-54.286,179.905,7.436,149.423
C06138=1122.244,62.845,-54.300,179.906,7.440,149.424
C06139=1122.240,63.060,-54.314,179.907,7.443,149.424
C06140=1122.235,63.310,-54.332,179.908,7.447,149.425
C06141=1122.230,63.559,-54.348,179.909,7.451,149.425
C06142=1122.225,63.808,-54.365,179.911,7.455,149.426
C06143=1122.220,64.058,-54.382,179.912,7.459,149.426
C06144=1122.215,64.308,-54.398,179.914,7.463,149.427
C06145=1122.210,64.557,-54.415,179.915,7.467,149.427
C06146=1122.205,64.806,-54.432,179.917,7.471,149.428
C06147=1122.201,65.055,-54.449,179.918,7.475,149.428
C06148=1122.196,65.305,-54.467,179.919,7.479,149.429
C06149=1122.191,65.554,-54.483,179.921,7.483,149.429
C06150=1122.185,65.803,-54.500,179.922,7.487,149.430
C06151=1122.181,66.053,-54.517,179.923,7.490,149.430
C06152=1122.176,66.303,-54.534,179.925,7.494,149.431
C06153=1122.171,66.551,-54.550,179.926,7.498,149.431
C06154=1122.165,66.801,-54.568,179.927,7.502,149.432
C06155=1122.161,67.050,-54.585,179.929,7.506,149.432
C06156=1122.156,67.300,-54.602,179.930,7.511,149.433
C06157=1122.151,67.549,-54.619,179.931,7.515,149.433
C06158=1122.146,67.799,-54.636,179.933,7.518,149.434
C06159=1122.141,68.048,-54.653,179.934,7.523,149.434
C06160=1122.136,68.297,-54.671,179.936,7.527,149.435
C06161=1122.132,68.547,-54.687,179.937,7.531,149.435
C06162=1122.126,68.796,-54.704,179.939,7.534,149.436
C06163=1122.122,69.045,-54.721,179.940,7.539,149.436
C06164=1122.117,69.294,-54.739,179.942,7.543,149.437
C06165=1122.112,69.544,-54.755,179.943,7.547,149.437
C06166=1122.107,69.794,-54.773,179.944,7.551,149.438
C06167=1122.102,70.044,-54.790,179.945,7.554,149.438
C06168=1122.097,70.292,-54.807,179.947,7.558,149.439
C06169=1122.092,70.541,-54.824,179.948,7.562,149.439
C06170=1122.087,70.791,-54.841,179.949,7.566,149.440
C06171=1122.082,71.040,-54.859,179.951,7.570,149.440
C06172=1122.077,71.290,-54.876,179.953,7.574,149.440
C06173=1122.073,71.539,-54.893,179.954,7.578,149.441
C06174=1122.068,71.789,-54.911,179.955,7.582,149.442
C06175=1122.063,72.037,-54.927,179.957,7.586,149.442
C06176=1122.058,72.287,-54.945,179.958,7.590,149.442
C06177=1122.053,72.536,-54.962,179.960,7.594,149.443
C06178=1122.048,72.786,-54.979,179.961,7.598,149.444
C06179=1122.043,73.035,-54.997,179.963,7.602,149.444
C06180=1122.038,73.285,-55.014,179.964,7.606,149.445
C06181=1122.034,73.534,-55.032,179.965,7.610,149.445
C06182=1122.028,73.783,-55.049,179.967,7.614,149.445
C06183=1122.024,74.033,-55.067,179.969,7.618,149.446
C06184=1122.018,74.282,-55.084,179.970,7.622,149.447
C06185=1122.014,74.531,-55.101,179.971,7.626,149.447
C06186=1122.008,74.780,-55.118,179.973,7.630,149.447
C06187=1122.003,75.030,-55.136,179.974,7.633,149.448
C06188=1122.000,75.245,-55.151,179.975,7.637,149.448
C06189=1121.996,75.459,-55.166,179.976,7.640,149.449
C06190=1121.992,75.674,-55.181,179.978,7.644,149.449
C06191=1121.987,75.888,-55.196,179.979,7.647,149.450
C06192=1121.983,76.103,-55.212,179.980,7.651,149.450
C06193=1121.978,76.318,-55.226,179.981,7.654,149.450
C06194=1121.974,76.533,-55.242,179.982,7.657,149.451
C06195=1121.970,76.747,-55.256,179.984,7.661,149.451
C06196=1121.965,76.996,-55.274,179.985,7.664,149.452
C06197=1121.960,77.246,-55.291,179.986,7.669,149.452
C06198=1121.955,77.495,-55.309,179.986,7.672,149.453
C06199=1121.950,77.744,-55.327,179.987,7.675,149.453
C06200=1121.946,77.993,-55.344,179.989,7.679,149.454
C06201=1121.941,78.243,-55.362,179.990,7.683,149.454
C06202=1121.936,78.492,-55.380,179.991,7.687,149.455
C06203=1121.931,78.742,-55.397,179.992,7.690,149.456
C06204=1121.926,78.991,-55.415,179.993,7.694,149.456
C06205=1121.921,79.240,-55.433,179.994,7.697,149.457
C06206=1121.916,79.489,-55.450,179.995,7.702,149.457
C06207=1121.911,79.739,-55.468,179.995,7.705,149.458
C06208=1121.907,79.988,-55.486,179.997,7.709,149.458
C06209=1121.901,80.237,-55.503,179.997,7.713,149.459
C06210=1121.896,80.487,-55.521,179.999,7.716,149.459
C06211=1121.891,80.736,-55.539,-180.000,7.721,149.460
C06212=1121.887,80.985,-55.557,-179.999,7.724,149.460
C06213=1121.881,81.235,-55.574,-179.998,7.728,149.461
C06214=1121.877,81.485,-55.593,-179.997,7.731,149.462
C06215=1121.873,81.734,-55.610,-179.996,7.736,149.462
C06216=1121.868,81.983,-55.628,-179.994,7.739,149.463
C06217=1121.863,82.232,-55.646,-179.993,7.743,149.463
C06218=1121.858,82.482,-55.663,-179.992,7.747,149.464
C06219=1121.853,82.731,-55.681,-179.991,7.750,149.464
C06220=1121.848,82.980,-55.699,-179.990,7.754,149.465
C06221=1121.843,83.229,-55.717,-179.988,7.758,149.465
C06222=1121.838,83.478,-55.735,-179.988,7.762,149.466
C06223=1121.833,83.728,-55.753,-179.986,7.766,149.466
C06224=1121.828,83.977,-55.770,-179.985,7.769,149.467
C06225=1121.823,84.227,-55.788,-179.984,7.773,149.467
C06226=1121.818,84.476,-55.806,-179.983,7.777,149.468
C06227=1121.814,84.726,-55.825,-179.981,7.781,149.468
C06228=1121.809,84.975,-55.843,-179.980,7.784,149.469
C06229=1121.804,85.224,-55.861,-179.979,7.788,149.469
C06230=1121.799,85.473,-55.879,-179.978,7.792,149.470
C06231=1121.794,85.722,-55.897,-179.976,7.796,149.470
C06232=1121.789,85.971,-55.915,-179.975,7.799,149.471
C06233=1121.784,86.221,-55.933,-179.974,7.804,149.471
C06234=1121.780,86.470,-55.951,-179.972,7.808,149.472
C06235=1121.775,86.720,-55.969,-179.971,7.811,149.472
C06236=1121.770,86.969,-55.987,-179.970,7.815,149.473
C06237=1121.765,87.218,-56.005,-179.969,7.819,149.473
C06238=1121.760,87.467,-56.023,-179.967,7.823,149.474
C06239=1121.756,87.716,-56.041,-179.966,7.827,149.474
C06240=1121.751,87.966,-56.059,-179.964,7.831,149.475
C06241=1121.746,88.215,-56.077,-179.963,7.834,149.475
C06242=1121.741,88.465,-56.096,-179.962,7.838,149.476
C06243=1121.736,88.714,-56.114,-179.961,7.842,149.476
C06244=1121.732,88.929,-56.129,-179.959,7.845,149.477
C06245=1121.728,89.143,-56.145,-179.958,7.849,149.477
C06246=1121.724,89.358,-56.161,-179.957,7.852,149.477
C06247=1121.720,89.572,-56.176,-179.956,7.855,149.478
C06248=1121.715,89.787,-56.191,-179.954,7.859,149.478
C06249=1121.710,90.001,-56.208,-179.953,7.862,149.479
C06250=1121.706,90.216,-56.223,-179.952,7.865,149.479
C06251=1121.702,90.430,-56.239,-179.951,7.869,149.480
C06252=1121.698,90.680,-56.258,-179.949,7.873,149.480
C06253=1121.693,90.929,-56.276,-179.947,7.877,149.480
C06254=1121.688,91.178,-56.294,-179.946,7.880,149.481
C06255=1121.683,91.427,-56.312,-179.945,7.884,149.481
C06256=1121.678,91.677,-56.330,-179.943,7.888,149.482
C06257=1121.674,91.926,-56.349,-179.942,7.892,149.482
C06258=1121.669,92.175,-56.367,-179.940,7.896,149.483
C06259=1121.664,92.424,-56.385,-179.939,7.900,149.483
C06260=1121.659,92.674,-56.404,-179.937,7.904,149.484
C06261=1121.654,92.924,-56.422,-179.936,7.908,149.484
C06262=1121.649,93.172,-56.441,-179.934,7.911,149.485
C06263=1121.644,93.421,-56.459,-179.933,7.915,149.485
C06264=1121.639,93.671,-56.478,-179.931,7.919,149.485
C06265=1121.635,93.920,-56.496,-179.929,7.923,149.486
C06266=1121.630,94.169,-56.514,-179.928,7.927,149.486
C06267=1121.625,94.418,-56.532,-179.926,7.931,149.487
C06268=1121.620,94.668,-56.552,-179.925,7.935,149.487
C06269=1121.615,94.917,-56.570,-179.923,7.939,149.488
C06270=1121.610,95.166,-56.588,-179.921,7.943,149.488
C06271=1121.606,95.416,-56.608,-179.920,7.946,149.488
C06272=1121.601,95.665,-56.626,-179.918,7.950,149.489
C06273=1121.596,95.914,-56.644,-179.917,7.954,149.489
C06274=1121.591,96.164,-56.663,-179.914,7.958,149.489
C06275=1121.586,96.413,-56.681,-179.913,7.962,149.490
C06276=1121.581,96.661,-56.700,-179.911,7.966,149.490
C06277=1121.576,96.912,-56.719,-179.910,7.969,149.491
C06278=1121.571,97.161,-56.737,-179.907,7.974,149.491
C06279=1121.567,97.409,-56.755,-179.906,7.978,149.492
C06280=1121.562,97.660,-56.774,-179.904,7.982,149.492
C06281=1121.557,97.908,-56.793,-179.902,7.985,149.492
C06282=1121.552,98.158,-56.812,-179.901,7.989,149.493
C06283=1121.548,98.407,-56.831,-179.899,7.993,149.493
C06284=1121.543,98.656,-56.849,-179.897,7.997,149.494
C06285=1121.538,98.906,-56.868,-179.895,8.001,149.494
C06286=1121.533,99.154,-56.887,-179.894,8.004,149.494
C06287=1121.528,99.404,-56.906,-179.891,8.009,149.495
C06288=1121.524,99.653,-56.925,-179.890,8.013,149.495
C06289=1121.518,99.902,-56.943,-179.888,8.016,149.495
C06290=1121.514,100.152,-56.962,-179.886,8.020,149.496
C06291=1121.508,100.401,-56.981,-179.885,8.024,149.496
C06292=1121.504,100.650,-57.000,-179.883,8.028,149.496
C06293=1121.499,100.899,-57.019,-179.880,8.032,149.497
C06294=1121.494,101.148,-57.037,-179.879,8.036,149.497
C06295=1121.489,101.398,-57.057,-179.877,8.040,149.497
C06296=1121.485,101.647,-57.076,-179.875,8.044,149.498
C06297=1121.480,101.897,-57.095,-179.873,8.047,149.498
C06298=1121.475,102.145,-57.113,-179.871,8.052,149.499
C06299=1121.470,102.395,-57.133,-179.869,8.055,149.499
C06300=1121.467,102.609,-57.149,-179.867,8.059,149.499
C06301=1121.462,102.824,-57.165,-179.866,8.062,149.499
C06302=1121.458,103.038,-57.181,-179.864,8.065,149.500
C06303=1121.453,103.253,-57.198,-179.863,8.069,149.500
C06304=1121.449,103.467,-57.214,-179.861,8.072,149.500
C06305=1121.445,103.681,-57.231,-179.859,8.076,149.500
C06306=1121.442,103.896,-57.247,-179.857,8.078,149.501
C06307=1121.437,104.110,-57.264,-179.856,8.082,149.501
C06308=1121.433,104.359,-57.282,-179.853,8.086,149.501
C06309=1121.427,104.609,-57.301,-179.851,8.090,149.502
C06310=1121.422,104.858,-57.321,-179.849,8.094,149.502
C06311=1121.418,105.107,-57.340,-179.847,8.097,149.502
C06312=1121.413,105.356,-57.359,-179.845,8.102,149.503
C06313=1121.409,105.605,-57.378,-179.843,8.106,149.503
C06314=1121.403,105.854,-57.397,-179.841,8.109,149.503
C06315=1121.399,106.104,-57.417,-179.839,8.113,149.504
C06316=1121.394,106.354,-57.435,-179.836,8.117,149.504
C06317=1121.389,106.602,-57.455,-179.834,8.121,149.504
C06318=1121.384,106.852,-57.474,-179.832,8.124,149.504
C06319=1121.379,107.101,-57.494,-179.830,8.129,149.505
C06320=1121.375,107.350,-57.513,-179.828,8.132,149.505
C06321=1121.370,107.599,-57.532,-179.826,8.136,149.505
C06322=1121.365,107.849,-57.552,-179.823,8.140,149.505
C06323=1121.361,108.098,-57.571,-179.821,8.144,149.506
C06324=1121.355,108.347,-57.590,-179.819,8.148,149.506
C06325=1121.351,108.596,-57.610,-179.817,8.152,149.506
C06326=1121.345,108.845,-57.629,-179.815,8.155,149.506
C06327=1121.341,109.094,-57.648,-179.812,8.160,149.507
C06328=1121.337,109.344,-57.668,-179.810,8.163,149.507
C06329=1121.331,109.593,-57.687,-179.808,8.167,149.507
C06330=1121.327,109.842,-57.707,-179.805,8.171,149.507
C06331=1121.322,110.091,-57.727,-179.803,8.174,149.508
C06332=1121.318,110.340,-57.746,-179.801,8.179,149.508
C06333=1121.313,110.590,-57.765,-179.799,8.182,149.508
C06334=1121.307,110.838,-57.785,-179.797,8.186,149.508
C06335=1121.303,111.088,-57.804,-179.794,8.190,149.508
C06336=1121.298,111.338,-57.824,-179.792,8.193,149.509
C06337=1121.293,111.586,-57.843,-179.791,8.197,149.509
C06338=1121.288,111.835,-57.864,-179.789,8.200,149.509
C06339=1121.284,112.085,-57.883,-179.787,8.204,149.510
C06340=1121.279,112.333,-57.902,-179.785,8.207,149.510
C06341=1121.274,112.583,-57.922,-179.783,8.211,149.510
C06342=1121.270,112.832,-57.942,-179.781,8.214,149.510
C06343=1121.265,113.082,-57.962,-179.779,8.218,149.511
C06344=1121.260,113.330,-57.981,-179.777,8.222,149.511
C06345=1121.255,113.580,-58.001,-179.776,8.225,149.511
C06346=1121.250,113.829,-58.021,-179.774,8.228,149.511
C06347=1121.245,114.078,-58.040,-179.772,8.232,149.512
C06348=1121.240,114.327,-58.060,-179.770,8.235,149.512
C06349=1121.236,114.576,-58.080,-179.768,8.239,149.512
C06350=1121.231,114.826,-58.100,-179.766,8.242,149.513
C06351=1121.226,115.075,-58.119,-179.764,8.246,149.513
C06352=1121.221,115.324,-58.140,-179.763,8.249,149.513
C06353=1121.217,115.573,-58.159,-179.761,8.253,149.513
C06354=1121.212,115.823,-58.179,-179.759,8.256,149.514
C06355=1121.207,116.071,-58.199,-179.757,8.260,149.514
C06356=1121.203,116.286,-58.216,-179.755,8.262,149.514
C06357=1121.199,116.500,-58.233,-179.754,8.265,149.514
C06358=1121.195,116.714,-58.249,-179.752,8.268,149.515
C06359=1121.191,116.929,-58.267,-179.750,8.271,149.515
C06360=1121.187,117.143,-58.284,-179.749,8.274,149.515
C06361=1121.183,117.357,-58.302,-179.748,8.277,149.515
C06362=1121.178,117.572,-58.318,-179.746,8.280,149.516
C06363=1121.174,117.786,-58.336,-179.744,8.283,149.516
C06364=1121.169,118.035,-58.355,-179.742,8.287,149.516
C06365=1121.165,118.284,-58.376,-179.740,8.290,149.516
C06366=1121.160,118.534,-58.395,-179.739,8.293,149.517
C06367=1121.156,118.783,-58.416,-179.737,8.297,149.517
C06368=1121.150,119.032,-58.435,-179.735,8.300,149.517
C06369=1121.146,119.281,-58.456,-179.733,8.304,149.517
C06370=1121.141,119.530,-58.475,-179.732,8.306,149.518
C06371=1121.136,119.779,-58.496,-179.730,8.310,149.518
C06372=1121.131,120.029,-58.516,-179.728,8.314,149.518
C06373=1121.127,120.278,-58.536,-179.726,8.317,149.519
C06374=1121.122,120.527,-58.556,-179.724,8.321,149.519
C06375=1121.117,120.776,-58.576,-179.722,8.324,149.519
C06376=1121.113,121.025,-58.596,-179.721,8.327,149.519
C06377=1121.108,121.274,-58.616,-179.719,8.331,149.520
C06378=1121.103,121.523,-58.637,-179.717,8.334,149.520
C06379=1121.098,121.772,-58.657,-179.715,8.337,149.520
C06380=1121.094,122.022,-58.677,-179.713,8.341,149.520
C06381=1121.089,122.271,-58.697,-179.712,8.345,149.521
C06382=1121.085,122.520,-58.718,-179.710,8.347,149.521
C06383=1121.079,122.769,-58.737,-179.708,8.351,149.521
C06384=1121.074,123.018,-58.758,-179.706,8.354,149.521
C06385=1121.070,123.267,-58.778,-179.704,8.358,149.522
C06386=1121.065,123.517,-58.798,-179.703,8.361,149.522
C06387=1121.061,123.765,-58.818,-179.701,8.364,149.522
C06388=1121.055,124.015,-58.839,-179.699,8.368,149.523
C06389=1121.051,124.264,-58.860,-179.697,8.371,149.523
C06390=1121.046,124.513,-58.879,-179.696,8.374,149.523
C06391=1121.042,124.762,-58.900,-179.694,8.378,149.523
C06392=1121.037,125.011,-58.921,-179.692,8.381,149.524
C06393=1121.032,125.260,-58.941,-179.690,8.384,149.524
C06394=1121.028,125.509,-58.961,-179.689,8.388,149.524
C06395=1121.023,125.759,-58.981,-179.686,8.392,149.525
C06396=1121.018,126.008,-59.002,-179.685,8.394,149.525
C06397=1121.013,126.257,-59.022,-179.683,8.398,149.525
C06398=1121.009,126.506,-59.043,-179.681,8.402,149.525
C06399=1121.004,126.755,-59.064,-179.680,8.404,149.526
C06400=1120.999,127.004,-59.084,-179.678,8.408,149.526
C06401=1120.995,127.253,-59.104,-179.676,8.411,149.526
C06402=1120.990,127.503,-59.125,-179.675,8.414,149.527
C06403=1120.985,127.752,-59.145,-179.673,8.418,149.527
C06404=1120.981,128.001,-59.165,-179.671,8.421,149.527
C06405=1120.975,128.250,-59.186,-179.669,8.424,149.527
C06406=1120.971,128.499,-59.207,-179.668,8.428,149.528
C06407=1120.966,128.749,-59.228,-179.665,8.431,149.528
C06408=1120.961,128.997,-59.248,-179.664,8.434,149.528
C06409=1120.957,129.246,-59.268,-179.662,8.438,149.528
C06410=1120.952,129.496,-59.289,-179.660,8.442,149.529
C06411=1120.947,129.745,-59.310,-179.659,8.444,149.529
C06412=1120.943,129.958,-59.327,-179.657,8.447,149.529
C06413=1120.939,130.173,-59.346,-179.655,8.450,149.529
C06414=1120.934,130.387,-59.363,-179.654,8.453,149.530
C06415=1120.931,130.601,-59.381,-179.652,8.456,149.530
C06416=1120.926,130.815,-59.398,-179.651,8.459,149.530
C06417=1120.922,131.030,-59.417,-179.650,8.461,149.530
C06418=1120.918,131.245,-59.434,-179.649,8.464,149.531
C06419=1120.914,131.458,-59.452,-179.647,8.467,149.531
C06420=1120.909,131.707,-59.473,-179.645,8.471,149.531
C06421=1120.905,131.956,-59.494,-179.643,8.474,149.531
C06422=1120.900,132.205,-59.515,-179.642,8.477,149.532
C06423=1120.896,132.455,-59.535,-179.640,8.481,149.532
C06424=1120.891,132.704,-59.556,-179.638,8.484,149.532
C06425=1120.886,132.953,-59.577,-179.636,8.487,149.533
C06426=1120.881,133.202,-59.598,-179.635,8.491,149.533
C06427=1120.877,133.451,-59.618,-179.633,8.494,149.533
C06428=1120.872,133.700,-59.640,-179.631,8.497,149.533
C06429=1120.867,133.949,-59.660,-179.630,8.501,149.534
C06430=1120.862,134.198,-59.681,-179.628,8.504,149.534
C06431=1120.858,134.447,-59.702,-179.626,8.507,149.534
C06432=1120.853,134.696,-59.723,-179.625,8.510,149.535
C06433=1120.849,134.945,-59.744,-179.623,8.514,149.535
C06434=1120.844,135.195,-59.765,-179.621,8.518,149.535
C06435=1120.839,135.444,-59.786,-179.620,8.520,149.536
C06436=1120.834,135.693,-59.806,-179.618,8.524,149.536
C06437=1120.829,135.941,-59.828,-179.617,8.527,149.536
C06438=1120.825,136.190,-59.848,-179.615,8.530,149.537
C06439=1120.820,136.440,-59.869,-179.613,8.534,149.537
C06440=1120.815,136.689,-59.891,-179.612,8.537,149.537
C06441=1120.811,136.938,-59.912,-179.610,8.540,149.537
C06442=1120.806,137.187,-59.933,-179.609,8.544,149.538
C06443=1120.801,137.436,-59.953,-179.607,8.547,149.538
C06444=1120.797,137.685,-59.975,-179.605,8.550,149.538
C06445=1120.792,137.935,-59.996,-179.603,8.554,149.539
C06446=1120.788,138.183,-60.017,-179.601,8.557,149.539
C06447=1120.783,138.432,-60.038,-179.600,8.560,149.539
C06448=1120.777,138.682,-60.059,-179.598,8.564,149.540
C06449=1120.773,138.930,-60.080,-179.596,8.567,149.540
C06450=1120.769,139.180,-60.102,-179.595,8.570,149.540
C06451=1120.764,139.429,-60.123,-179.593,8.574,149.541
C06452=1120.759,139.678,-60.144,-179.592,8.577,149.541
C06453=1120.754,139.927,-60.165,-179.590,8.580,149.541
C06454=1120.749,140.175,-60.186,-179.589,8.583,149.542
C06455=1120.745,140.425,-60.208,-179.587,8.587,149.542
C06456=1120.741,140.674,-60.229,-179.585,8.591,149.542
C06457=1120.736,140.923,-60.250,-179.584,8.593,149.543
C06458=1120.731,141.172,-60.271,-179.582,8.597,149.543
C06459=1120.726,141.422,-60.293,-179.581,8.600,149.543
C06460=1120.722,141.670,-60.314,-179.579,8.604,149.544
C06461=1120.717,141.919,-60.335,-179.578,8.607,149.544
C06462=1120.713,142.169,-60.357,-179.576,8.610,149.544
C06463=1120.707,142.418,-60.378,-179.575,8.613,149.545
C06464=1120.703,142.666,-60.399,-179.573,8.617,149.545
C06465=1120.698,142.915,-60.420,-179.571,8.621,149.545
C06466=1120.694,143.165,-60.442,-179.570,8.624,149.546
C06467=1120.689,143.413,-60.463,-179.568,8.627,149.546
C06468=1120.685,143.628,-60.481,-179.567,8.630,149.546
C06469=1120.681,143.841,-60.500,-179.565,8.633,149.547
C06470=1120.677,144.056,-60.518,-179.564,8.636,149.547
C06471=1120.673,144.270,-60.537,-179.563,8.639,149.547
C06472=1120.669,144.484,-60.555,-179.561,8.641,149.547
C06473=1120.664,144.698,-60.573,-179.560,8.645,149.548
C06474=1120.660,144.912,-60.592,-179.559,8.647,149.548
C06475=1120.657,145.127,-60.610,-179.558,8.650,149.548
C06476=1120.652,145.375,-60.632,-179.555,8.654,149.549
C06477=1120.648,145.625,-60.654,-179.553,8.658,149.549
C06478=1120.642,145.874,-60.675,-179.550,8.662,149.549
C06479=1120.638,146.123,-60.697,-179.548,8.665,149.549
C06480=1120.633,146.372,-60.719,-179.545,8.670,149.549
C06481=1120.628,146.621,-60.740,-179.543,8.673,149.550
C06482=1120.624,146.869,-60.761,-179.541,8.677,149.550
C06483=1120.620,147.119,-60.783,-179.538,8.681,149.550
C06484=1120.615,147.367,-60.804,-179.536,8.684,149.550
C06485=1120.610,147.617,-60.825,-179.534,8.689,149.551
C06486=1120.605,147.866,-60.847,-179.532,8.692,149.551
C06487=1120.601,148.115,-60.869,-179.529,8.695,149.551
C06488=1120.596,148.364,-60.891,-179.526,8.700,149.551
C06489=1120.591,148.613,-60.913,-179.524,8.703,149.551
C06490=1120.587,148.861,-60.935,-179.522,8.707,149.552
C06491=1120.582,149.111,-60.956,-179.519,8.711,149.552
C06492=1120.577,149.360,-60.978,-179.517,8.714,149.552
C06493=1120.573,149.609,-61.000,-179.514,8.718,149.552
C06494=1120.568,149.858,-61.021,-179.512,8.722,149.552
C06495=1120.564,150.107,-61.043,-179.510,8.725,149.553
C06496=1120.559,150.356,-61.065,-179.507,8.729,149.553
C06497=1120.554,150.605,-61.087,-179.505,8.733,149.553
C06498=1120.549,150.854,-61.109,-179.503,8.736,149.553
C06499=1120.544,151.103,-61.131,-179.501,8.740,149.553
C06500=1120.540,151.352,-61.153,-179.498,8.744,149.554
C06501=1120.535,151.601,-61.175,-179.495,8.747,149.554
C06502=1120.531,151.850,-61.197,-179.493,8.750,149.554
C06503=1120.526,152.099,-61.218,-179.491,8.754,149.554
C06504=1120.522,152.348,-61.241,-179.488,8.758,149.554
C06505=1120.517,152.597,-61.262,-179.486,8.761,149.554
C06506=1120.512,152.846,-61.284,-179.484,8.765,149.555
C06507=1120.507,153.095,-61.307,-179.481,8.768,149.555
C06508=1120.503,153.344,-61.329,-179.479,8.772,149.555
C06509=1120.498,153.593,-61.350,-179.476,8.775,149.555
C06510=1120.494,153.842,-61.373,-179.474,8.779,149.555
C06511=1120.489,154.090,-61.395,-179.472,8.782,149.555
C06512=1120.485,154.340,-61.417,-179.470,8.785,149.555
C06513=1120.479,154.589,-61.439,-179.467,8.789,149.556
C06514=1120.475,154.838,-61.461,-179.464,8.793,149.556
C06515=1120.470,155.087,-61.483,-179.462,8.796,149.556
C06516=1120.466,155.335,-61.506,-179.460,8.800,149.556
C06517=1120.460,155.584,-61.528,-179.458,8.803,149.556
C06518=1120.456,155.834,-61.550,-179.455,8.806,149.556
C06519=1120.452,156.083,-61.572,-179.453,8.809,149.556
C06520=1120.447,156.331,-61.594,-179.451,8.813,149.557
C06521=1120.442,156.581,-61.617,-179.448,8.817,149.557
C06522=1120.437,156.829,-61.639,-179.446,8.820,149.557
C06523=1120.433,157.079,-61.661,-179.443,8.823,149.557
C06524=1120.429,157.292,-61.680,-179.442,8.826,149.557
C06525=1120.425,157.506,-61.700,-179.439,8.829,149.557
C06526=1120.421,157.721,-61.719,-179.438,8.832,149.557
C06527=1120.417,157.935,-61.738,-179.435,8.835,149.557
C06528=1120.413,158.149,-61.757,-179.433,8.837,149.558
C06529=1120.409,158.363,-61.777,-179.431,8.841,149.558
C06530=1120.405,158.577,-61.796,-179.429,8.843,149.558
C06531=1120.401,158.791,-61.815,-179.427,8.847,149.558
C06532=1120.396,159.040,-61.836,-179.425,8.850,149.558
C06533=1120.392,159.288,-61.859,-179.423,8.853,149.558
C06534=1120.387,159.538,-61.882,-179.420,8.856,149.558
C06535=1120.383,159.786,-61.904,-179.418,8.859,149.558
C06536=1120.378,160.036,-61.927,-179.415,8.863,149.559
C06537=1120.374,160.284,-61.950,-179.413,8.866,149.559
C06538=1120.369,160.533,-61.971,-179.411,8.870,149.559
C06539=1120.364,160.782,-61.995,-179.408,8.873,149.559
C06540=1120.360,161.031,-62.017,-179.406,8.876,149.559
C06541=1120.354,161.280,-62.040,-179.404,8.879,149.559
C06542=1120.350,161.529,-62.062,-179.401,8.882,149.559
C06543=1120.346,161.778,-62.085,-179.399,8.886,149.559
C06544=1120.341,162.027,-62.107,-179.397,8.889,149.559
C06545=1120.337,162.275,-62.130,-179.394,8.892,149.559
C06546=1120.332,162.525,-62.152,-179.392,8.896,149.560
C06547=1120.328,162.774,-62.175,-179.390,8.899,149.560
C06548=1120.322,163.022,-62.198,-179.388,8.901,149.560
C06549=1120.318,163.271,-62.220,-179.386,8.904,149.560
C06550=1120.313,163.520,-62.243,-179.383,8.908,149.560
C06551=1120.309,163.770,-62.265,-179.381,8.911,149.560
C06552=1120.304,164.018,-62.288,-179.378,8.914,149.560
C06553=1120.300,164.267,-62.311,-179.376,8.917,149.560
C06554=1120.295,164.517,-62.334,-179.374,8.921,149.561
C06555=1120.291,164.765,-62.357,-179.371,8.924,149.561
C06556=1120.286,165.014,-62.380,-179.369,8.927,149.561
C06557=1120.282,165.262,-62.402,-179.367,8.930,149.561
C06558=1120.277,165.512,-62.425,-179.365,8.933,149.561
C06559=1120.272,165.761,-62.448,-179.362,8.936,149.561
C06560=1120.268,166.010,-62.471,-179.360,8.939,149.561
C06561=1120.262,166.259,-62.493,-179.358,8.942,149.561
C06562=1120.258,166.507,-62.516,-179.355,8.946,149.561
C06563=1120.254,166.756,-62.540,-179.353,8.949,149.562
C06564=1120.249,167.005,-62.563,-179.350,8.952,149.562
C06565=1120.245,167.254,-62.586,-179.349,8.954,149.562
C06566=1120.239,167.503,-62.608,-179.347,8.958,149.562
C06567=1120.235,167.752,-62.631,-179.344,8.961,149.562
C06568=1120.231,168.001,-62.654,-179.341,8.964,149.562
C06569=1120.226,168.250,-62.677,-179.339,8.967,149.562
C06570=1120.221,168.499,-62.701,-179.337,8.970,149.562
C06571=1120.217,168.748,-62.724,-179.335,8.973,149.562
C06572=1120.212,168.996,-62.747,-179.332,8.976,149.562
C06573=1120.207,169.245,-62.770,-179.330,8.980,149.562
C06574=1120.203,169.494,-62.792,-179.328,8.983,149.563
C06575=1120.198,169.743,-62.815,-179.326,8.985,149.563
C06576=1120.194,169.992,-62.839,-179.324,8.989,149.563
C06577=1120.189,170.241,-62.862,-179.321,8.992,149.563
C06578=1120.185,170.490,-62.885,-179.319,8.995,149.563
C06579=1120.180,170.738,-62.908,-179.317,8.997,149.563
C06580=1120.177,170.953,-62.928,-179.315,9.001,149.563
C06581=1120.172,171.167,-62.948,-179.313,9.003,149.563
C06582=1120.168,171.380,-62.968,-179.311,9.005,149.563
C06583=1120.164,171.594,-62.987,-179.309,9.008,149.563
C06584=1120.160,171.808,-63.008,-179.307,9.011,149.563
C06585=1120.157,172.023,-63.028,-179.305,9.013,149.564
C06586=1120.153,172.236,-63.048,-179.303,9.016,149.564
C06587=1120.148,172.450,-63.068,-179.301,9.018,149.564
C06588=1120.144,172.699,-63.091,-179.299,9.022,149.564
C06589=1120.140,172.948,-63.114,-179.297,9.025,149.564
C06590=1120.135,173.197,-63.138,-179.295,9.027,149.564
C06591=1120.130,173.446,-63.161,-179.293,9.031,149.564
C06592=1120.125,173.695,-63.184,-179.290,9.034,149.564
C06593=1120.122,173.944,-63.207,-179.288,9.036,149.564
C06594=1120.117,174.192,-63.231,-179.286,9.039,149.564
C06595=1120.112,174.441,-63.254,-179.284,9.043,149.564
C06596=1120.108,174.690,-63.278,-179.282,9.045,149.564
C06597=1120.103,174.939,-63.301,-179.279,9.048,149.565
C06598=1120.098,175.188,-63.325,-179.277,9.051,149.565
C06599=1120.093,175.436,-63.347,-179.275,9.054,149.565
C06600=1120.089,175.685,-63.372,-179.273,9.057,149.565
C06601=1120.085,175.934,-63.394,-179.271,9.060,149.565
C06602=1120.080,176.183,-63.418,-179.269,9.063,149.565
C06603=1120.075,176.432,-63.441,-179.266,9.066,149.565
C06604=1120.071,176.680,-63.465,-179.264,9.069,149.565
C06605=1120.066,176.929,-63.488,-179.262,9.072,149.565
C06606=1120.062,177.179,-63.512,-179.260,9.075,149.565
C06607=1120.057,177.428,-63.536,-179.258,9.078,149.566
C06608=1120.053,177.676,-63.560,-179.256,9.081,149.566
C06609=1120.048,177.925,-63.583,-179.253,9.084,149.566
C06610=1120.044,178.174,-63.606,-179.251,9.087,149.566
C06611=1120.039,178.423,-63.630,-179.249,9.090,149.566
C06612=1120.035,178.672,-63.654,-179.247,9.093,149.566
C06613=1120.030,178.921,-63.677,-179.245,9.095,149.566
C06614=1120.025,179.169,-63.701,-179.243,9.098,149.566
C06615=1120.021,179.418,-63.725,-179.240,9.102,149.566
C06616=1120.016,179.667,-63.749,-179.238,9.105,149.566
C06617=1120.012,179.916,-63.772,-179.235,9.109,149.567
C06618=1120.007,180.164,-63.796,-179.232,9.112,149.567
C06619=1120.003,180.413,-63.819,-179.230,9.115,149.567
C06620=1119.998,180.662,-63.843,-179.227,9.118,149.567
C06621=1119.993,180.911,-63.867,-179.224,9.121,149.566
C06622=1119.989,181.160,-63.890,-179.221,9.124,149.567
C06623=1119.985,181.409,-63.915,-179.218,9.128,149.567
C06624=1119.980,181.658,-63.938,-179.216,9.131,149.567
C06625=1119.976,181.906,-63.962,-179.213,9.134,149.567
C06626=1119.971,182.155,-63.985,-179.211,9.137,149.567
C06627=1119.966,182.404,-64.010,-179.208,9.140,149.567
C06628=1119.962,182.652,-64.034,-179.206,9.143,149.567
C06629=1119.957,182.901,-64.058,-179.203,9.146,149.567
C06630=1119.953,183.150,-64.082,-179.200,9.149,149.567
C06631=1119.948,183.400,-64.105,-179.198,9.152,149.567
C06632=1119.944,183.648,-64.129,-179.195,9.155,149.567
C06633=1119.939,183.897,-64.154,-179.193,9.158,149.567
C06634=1119.934,184.146,-64.177,-179.190,9.161,149.567
C06635=1119.930,184.394,-64.202,-179.188,9.165,149.567
C06636=1119.926,184.609,-64.222,-179.185,9.166,149.567
C06637=1119.922,184.822,-64.243,-179.183,9.169,149.567
C06638=1119.919,185.036,-64.264,-179.181,9.172,149.567
C06639=1119.914,185.249,-64.285,-179.179,9.174,149.567
C06640=1119.911,185.463,-64.305,-179.177,9.177,149.567
C06641=1119.907,185.678,-64.325,-179.175,9.180,149.567
C06642=1119.902,185.891,-64.346,-179.173,9.182,149.567
C06643=1119.899,186.105,-64.367,-179.171,9.184,149.567
C06644=1119.894,186.354,-64.391,-179.168,9.187,149.567
C06645=1119.890,186.602,-64.415,-179.166,9.191,149.567
C06646=1119.885,186.851,-64.439,-179.164,9.193,149.567
C06647=1119.881,187.100,-64.463,-179.161,9.196,149.567
C06648=1119.876,187.349,-64.488,-179.158,9.199,149.567
C06649=1119.872,187.598,-64.512,-179.157,9.201,149.567
C06650=1119.867,187.846,-64.536,-179.154,9.204,149.567
C06651=1119.863,188.095,-64.561,-179.151,9.207,149.567
C06652=1119.858,188.344,-64.585,-179.150,9.210,149.567
C06653=1119.854,188.593,-64.608,-179.147,9.213,149.567
C06654=1119.849,188.842,-64.633,-179.145,9.216,149.567
C06655=1119.845,189.091,-64.658,-179.143,9.218,149.567
C06656=1119.840,189.339,-64.682,-179.140,9.221,149.567
C06657=1119.835,189.588,-64.706,-179.138,9.224,149.567
C06658=1119.831,189.836,-64.730,-179.136,9.227,149.567
C06659=1119.826,190.086,-64.755,-179.134,9.229,149.567
C06660=1119.822,190.334,-64.779,-179.132,9.233,149.568
C06661=1119.817,190.582,-64.804,-179.130,9.235,149.568
C06662=1119.812,190.831,-64.828,-179.127,9.238,149.568
C06663=1119.809,191.080,-64.853,-179.125,9.240,149.568
C06664=1119.803,191.329,-64.877,-179.123,9.243,149.568
C06665=1119.799,191.577,-64.901,-179.121,9.246,149.568
C06666=1119.795,191.827,-64.926,-179.119,9.248,149.568
C06667=1119.790,192.075,-64.950,-179.117,9.252,149.568
C06668=1119.786,192.324,-64.975,-179.115,9.254,149.568
C06669=1119.781,192.573,-65.000,-179.113,9.257,149.568
C06670=1119.777,192.821,-65.024,-179.111,9.259,149.568
C06671=1119.772,193.070,-65.048,-179.109,9.262,149.568
C06672=1119.768,193.319,-65.073,-179.107,9.265,149.569
C06673=1119.763,193.568,-65.097,-179.105,9.267,149.569
C06674=1119.758,193.816,-65.122,-179.103,9.270,149.569
C06675=1119.754,194.066,-65.147,-179.101,9.273,149.569
C06676=1119.749,194.314,-65.171,-179.099,9.276,149.569
C06677=1119.744,194.563,-65.195,-179.097,9.278,149.569
C06678=1119.741,194.812,-65.220,-179.096,9.281,149.569
C06679=1119.736,195.060,-65.245,-179.093,9.284,149.569
C06680=1119.732,195.309,-65.270,-179.092,9.286,149.570
C06681=1119.727,195.558,-65.294,-179.090,9.289,149.570
C06682=1119.722,195.806,-65.318,-179.088,9.291,149.570
C06683=1119.718,196.056,-65.343,-179.086,9.294,149.570
C06684=1119.714,196.293,-65.367,-179.085,9.297,149.570
C06685=1119.709,196.532,-65.391,-179.082,9.300,149.570
C06686=1119.705,196.770,-65.415,-179.079,9.303,149.570
C06687=1119.700,197.008,-65.438,-179.075,9.307,149.570
C06688=1119.697,197.246,-65.462,-179.073,9.310,149.570
C06689=1119.691,197.484,-65.485,-179.069,9.313,149.570
C06690=1119.688,197.722,-65.509,-179.067,9.316,149.570
C06691=1119.683,197.961,-65.533,-179.063,9.320,149.570
C06692=1119.679,198.185,-65.556,-179.060,9.323,149.570
C06693=1119.676,198.410,-65.578,-179.057,9.326,149.570
C06694=1119.671,198.634,-65.600,-179.055,9.328,149.569
C06695=1119.667,198.858,-65.622,-179.052,9.332,149.570
C06696=1119.664,199.082,-65.645,-179.049,9.334,149.569
C06697=1119.659,199.306,-65.667,-179.047,9.337,149.569
C06698=1119.655,199.531,-65.691,-179.043,9.341,149.569
C06699=1119.651,199.755,-65.713,-179.040,9.344,149.569
C06700=1119.647,200.004,-65.737,-179.037,9.346,149.569
C06701=1119.642,200.252,-65.763,-179.034,9.350,149.569
C06702=1119.638,200.501,-65.788,-179.031,9.353,149.569
C06703=1119.633,200.749,-65.813,-179.028,9.356,149.569
C06704=1119.629,200.998,-65.838,-179.024,9.359,149.569
C06705=1119.624,201.247,-65.863,-179.022,9.362,149.569
C06706=1119.620,201.496,-65.888,-179.019,9.365,149.569
C06707=1119.616,201.744,-65.913,-179.015,9.369,149.568
C06708=1119.611,201.993,-65.938,-179.012,9.371,149.568
C06709=1119.606,202.241,-65.963,-179.009,9.374,149.568
C06710=1119.602,202.491,-65.988,-179.007,9.377,149.568
C06711=1119.598,202.739,-66.014,-179.003,9.381,149.568
C06712=1119.593,202.988,-66.038,-179.000,9.384,149.568
C06713=1119.589,203.237,-66.064,-178.997,9.386,149.568
C06714=1119.584,203.485,-66.089,-178.995,9.389,149.568
C06715=1119.580,203.734,-66.114,-178.992,9.392,149.568
C06716=1119.575,203.982,-66.140,-178.989,9.395,149.567
C06717=1119.571,204.231,-66.165,-178.985,9.398,149.567
C06718=1119.567,204.480,-66.190,-178.982,9.401,149.567
C06719=1119.562,204.728,-66.215,-178.980,9.404,149.567
C06720=1119.558,204.977,-66.241,-178.977,9.407,149.567
C06721=1119.553,205.226,-66.266,-178.974,9.410,149.567
C06722=1119.548,205.475,-66.291,-178.971,9.412,149.567
C06723=1119.544,205.723,-66.317,-178.969,9.416,149.567
C06724=1119.539,205.972,-66.342,-178.966,9.418,149.567
C06725=1119.535,206.220,-66.368,-178.963,9.421,149.567
C06726=1119.531,206.470,-66.393,-178.960,9.424,149.567
C06727=1119.526,206.718,-66.419,-178.957,9.427,149.566
C06728=1119.522,206.967,-66.444,-178.954,9.430,149.566
C06729=1119.517,207.216,-66.470,-178.952,9.433,149.566
C06730=1119.513,207.464,-66.496,-178.949,9.436,149.566
C06731=1119.508,207.713,-66.521,-178.946,9.438,149.566
C06732=1119.504,207.962,-66.546,-178.943,9.441,149.566
C06733=1119.499,208.210,-66.572,-178.941,9.443,149.566
C06734=1119.495,208.459,-66.597,-178.938,9.446,149.566
C06735=1119.491,208.708,-66.623,-178.935,9.449,149.566
C06736=1119.486,208.956,-66.649,-178.933,9.452,149.566
C06737=1119.481,209.204,-66.674,-178.930,9.455,149.566
C06738=1119.477,209.453,-66.700,-178.927,9.458,149.566
C06739=1119.472,209.701,-66.725,-178.925,9.461,149.566
C06740=1119.468,209.950,-66.751,-178.923,9.463,149.566
C06741=1119.464,210.199,-66.777,-178.920,9.466,149.566
C06742=1119.460,210.448,-66.803,-178.918,9.469,149.566
C06743=1119.455,210.696,-66.828,-178.915,9.472,149.566
C06744=1119.451,210.945,-66.854,-178.912,9.475,149.566
C06745=1119.446,211.194,-66.880,-178.910,9.478,149.566
C06746=1119.442,211.443,-66.906,-178.908,9.481,149.566
C06747=1119.437,211.691,-66.931,-178.905,9.484,149.566
C06748=1119.433,211.904,-66.954,-178.903,9.486,149.566
C06749=1119.430,212.118,-66.975,-178.901,9.488,149.566
C06750=1119.426,212.332,-66.998,-178.899,9.490,149.566
C06751=1119.422,212.545,-67.020,-178.897,9.494,149.566
C06752=1119.418,212.759,-67.042,-178.895,9.496,149.566
C06753=1119.414,212.972,-67.064,-178.893,9.498,149.566
C06754=1119.410,213.186,-67.087,-178.891,9.501,149.566
C06755=1119.407,213.399,-67.109,-178.889,9.503,149.566
C06756=1119.403,213.648,-67.135,-178.887,9.506,149.566
C06757=1119.398,213.897,-67.161,-178.885,9.509,149.567
C06758=1119.393,214.146,-67.187,-178.883,9.512,149.567
C06759=1119.389,214.394,-67.212,-178.881,9.515,149.567
C06760=1119.385,214.642,-67.239,-178.878,9.518,149.567
C06761=1119.380,214.891,-67.264,-178.877,9.520,149.567
C06762=1119.376,215.140,-67.291,-178.874,9.523,149.567
C06763=1119.371,215.389,-67.316,-178.873,9.526,149.567
C06764=1119.367,215.637,-67.342,-178.870,9.529,149.567
C06765=1119.363,215.885,-67.368,-178.869,9.532,149.568
C06766=1119.358,216.134,-67.395,-178.866,9.535,149.568
C06767=1119.353,216.383,-67.420,-178.864,9.538,149.568
C06768=1119.349,216.631,-67.447,-178.862,9.540,149.568
C06769=1119.345,216.880,-67.473,-178.860,9.544,149.568
C06770=1119.340,217.129,-67.499,-178.857,9.547,149.568
C06771=1119.336,217.377,-67.525,-178.856,9.549,149.568
C06772=1119.332,217.625,-67.551,-178.853,9.553,149.568
C06773=1119.327,217.874,-67.577,-178.850,9.556,149.568
C06774=1119.323,218.123,-67.604,-178.848,9.559,149.569
C06775=1119.318,218.371,-67.629,-178.846,9.561,149.569
C06776=1119.314,218.620,-67.655,-178.844,9.565,149.569
C06777=1119.310,218.869,-67.682,-178.841,9.568,149.569
C06778=1119.305,219.117,-67.708,-178.839,9.571,149.569
C06779=1119.301,219.366,-67.734,-178.837,9.574,149.569
C06780=1119.296,219.615,-67.761,-178.834,9.577,149.569
C06781=1119.292,219.863,-67.787,-178.832,9.580,149.569
C06782=1119.288,220.112,-67.814,-178.830,9.583,149.569
C06783=1119.283,220.360,-67.840,-178.827,9.586,149.569
C06784=1119.279,220.608,-67.865,-178.825,9.589,149.569
C06785=1119.274,220.857,-67.892,-178.822,9.592,149.570
C06786=1119.270,221.106,-67.918,-178.820,9.595,149.570
C06787=1119.265,221.354,-67.945,-178.817,9.598,149.570
C06788=1119.261,221.603,-67.971,-178.815,9.602,149.570
C06789=1119.257,221.851,-67.998,-178.813,9.605,149.570
C06790=1119.252,222.100,-68.024,-178.810,9.608,149.570
C06791=1119.248,222.348,-68.050,-178.808,9.611,149.570
C06792=1119.244,222.597,-68.077,-178.804,9.615,149.570
C06793=1119.239,222.846,-68.103,-178.801,9.618,149.570
C06794=1119.235,223.094,-68.130,-178.799,9.621,149.570
C06795=1119.230,223.343,-68.156,-178.796,9.624,149.570
C06796=1119.226,223.592,-68.183,-178.794,9.627,149.570
C06797=1119.222,223.840,-68.209,-178.791,9.630,149.570
C06798=1119.217,224.089,-68.236,-178.789,9.633,149.570
C06799=1119.213,224.337,-68.262,-178.786,9.637,149.571
C06800=1119.208,224.585,-68.289,-178.783,9.640,149.570
C06801=1119.204,224.834,-68.316,-178.780,9.643,149.570
C06802=1119.199,225.083,-68.342,-178.778,9.646,149.571
C06803=1119.195,225.331,-68.369,-178.775,9.649,149.571
C06804=1119.192,225.545,-68.391,-178.772,9.652,149.570
C06805=1119.188,225.758,-68.415,-178.770,9.655,149.571
C06806=1119.184,225.971,-68.438,-178.768,9.657,149.571
C06807=1119.180,226.185,-68.461,-178.765,9.660,149.570
C06808=1119.176,226.398,-68.484,-178.762,9.663,149.570
C06809=1119.173,226.612,-68.507,-178.760,9.666,149.571
C06810=1119.169,226.826,-68.529,-178.757,9.668,149.570
C06811=1119.165,227.039,-68.553,-178.755,9.672,149.570
C06812=1119.161,227.288,-68.579,-178.752,9.674,149.570
C06813=1119.157,227.536,-68.606,-178.749,9.678,149.570
C06814=1119.152,227.784,-68.633,-178.746,9.681,149.570
C06815=1119.147,228.033,-68.660,-178.743,9.685,149.570
C06816=1119.143,228.281,-68.686,-178.740,9.688,149.570
C06817=1119.139,228.530,-68.713,-178.737,9.690,149.570
C06818=1119.134,228.778,-68.740,-178.734,9.694,149.570
C06819=1119.130,229.027,-68.768,-178.731,9.697,149.570
C06820=1119.126,229.276,-68.794,-178.727,9.700,149.570
C06821=1119.121,229.524,-68.821,-178.724,9.703,149.570
C06822=1119.117,229.773,-68.848,-178.721,9.707,149.570
C06823=1119.113,230.021,-68.875,-178.718,9.710,149.570
C06824=1119.108,230.269,-68.902,-178.714,9.713,149.570
C06825=1119.104,230.518,-68.929,-178.711,9.716,149.570
C06826=1119.099,230.767,-68.956,-178.709,9.719,149.569
C06827=1119.095,231.015,-68.983,-178.705,9.722,149.569
C06828=1119.091,231.264,-69.010,-178.702,9.725,149.569
C06829=1119.086,231.512,-69.037,-178.699,9.728,149.569
C06830=1119.082,231.760,-69.065,-178.695,9.731,149.569
C06831=1119.077,232.008,-69.092,-178.693,9.734,149.569
C06832=1119.073,232.258,-69.119,-178.690,9.737,149.569
C06833=1119.069,232.506,-69.146,-178.687,9.740,149.569
C06834=1119.065,232.754,-69.173,-178.684,9.743,149.569
C06835=1119.060,233.003,-69.200,-178.681,9.746,149.569
C06836=1119.056,233.251,-69.228,-178.678,9.749,149.568
C06837=1119.052,233.500,-69.255,-178.675,9.752,149.568
C06838=1119.047,233.748,-69.282,-178.672,9.754,149.568
C06839=1119.042,233.997,-69.309,-178.669,9.757,149.568
C06840=1119.038,234.245,-69.337,-178.666,9.760,149.568
C06841=1119.035,234.494,-69.364,-178.663,9.763,149.568
C06842=1119.030,234.742,-69.391,-178.660,9.765,149.568
C06843=1119.026,234.990,-69.419,-178.657,9.768,149.568
C06844=1119.022,235.239,-69.446,-178.654,9.771,149.568
C06845=1119.017,235.488,-69.473,-178.652,9.773,149.567
C06846=1119.013,235.736,-69.501,-178.649,9.776,149.567
C06847=1119.008,235.984,-69.528,-178.646,9.779,149.567
C06848=1119.004,236.233,-69.555,-178.643,9.782,149.567
C06849=1118.999,236.481,-69.583,-178.640,9.784,149.567
C06850=1118.995,236.730,-69.610,-178.637,9.787,149.567
C06851=1118.991,236.978,-69.638,-178.636,9.789,149.567
C06852=1118.986,237.227,-69.665,-178.633,9.792,149.567
C06853=1118.982,237.475,-69.693,-178.630,9.795,149.567
C06854=1118.978,237.724,-69.721,-178.627,9.797,149.567
C06855=1118.974,237.972,-69.748,-178.624,9.800,149.566
C06856=1118.969,238.220,-69.775,-178.622,9.803,149.566
C06857=1118.965,238.469,-69.803,-178.620,9.805,149.566
C06858=1118.961,238.717,-69.831,-178.617,9.807,149.566
C06859=1118.956,238.965,-69.858,-178.614,9.810,149.566
C06860=1118.952,239.180,-69.882,-178.612,9.813,149.566
C06861=1118.948,239.393,-69.906,-178.609,9.814,149.566
C06862=1118.945,239.606,-69.929,-178.608,9.817,149.566
C06863=1118.941,239.820,-69.953,-178.605,9.819,149.566
C06864=1118.937,240.033,-69.977,-178.603,9.821,149.566
C06865=1118.933,240.246,-70.001,-178.601,9.823,149.566
C06866=1118.929,240.459,-70.024,-178.599,9.825,149.566
C06867=1118.926,240.673,-70.048,-178.597,9.827,149.566
C06868=1118.922,240.921,-70.076,-178.595,9.830,149.566
C06869=1118.918,241.169,-70.105,-178.592,9.832,149.566
C06870=1118.913,241.418,-70.132,-178.590,9.835,149.566
C06871=1118.909,241.666,-70.159,-178.588,9.837,149.566
C06872=1118.905,241.914,-70.188,-178.585,9.840,149.566
C06873=1118.900,242.163,-70.215,-178.583,9.842,149.566
C06874=1118.896,242.411,-70.243,-178.581,9.844,149.566
C06875=1118.892,242.659,-70.271,-178.578,9.847,149.565
C06876=1118.887,242.908,-70.298,-178.576,9.849,149.566
C06877=1118.883,243.157,-70.326,-178.574,9.852,149.566
C06878=1118.879,243.405,-70.354,-178.571,9.854,149.565
C06879=1118.875,243.653,-70.382,-178.569,9.857,149.566
C06880=1118.870,243.902,-70.409,-178.568,9.859,149.566
C06881=1118.866,244.151,-70.438,-178.566,9.861,149.566
C06882=1118.861,244.398,-70.466,-178.563,9.864,149.566
C06883=1118.858,244.647,-70.494,-178.561,9.866,149.566
C06884=1118.853,244.895,-70.522,-178.559,9.869,149.566
C06885=1118.848,245.144,-70.549,-178.557,9.871,149.566
C06886=1118.844,245.392,-70.578,-178.555,9.873,149.566
C06887=1118.840,245.640,-70.605,-178.553,9.876,149.566
C06888=1118.836,245.889,-70.633,-178.551,9.879,149.566
C06889=1118.831,246.137,-70.662,-178.549,9.881,149.566
C06890=1118.827,246.385,-70.690,-178.547,9.884,149.566
C06891=1118.822,246.634,-70.717,-178.545,9.886,149.566
C06892=1118.818,246.883,-70.746,-178.544,9.889,149.566
C06893=1118.814,247.131,-70.774,-178.542,9.891,149.566
C06894=1118.810,247.379,-70.802,-178.540,9.893,149.566
C06895=1118.805,247.627,-70.829,-178.536,9.897,149.566
C06896=1118.801,247.876,-70.858,-178.531,9.902,149.566
C06897=1118.797,248.124,-70.886,-178.526,9.905,149.566
C06898=1118.792,248.373,-70.915,-178.522,9.909,149.566
C06899=1118.788,248.621,-70.943,-178.517,9.913,149.565
C06900=1118.784,248.869,-70.971,-178.512,9.917,149.565
C06901=1118.779,249.117,-70.999,-178.508,9.921,149.565
C06902=1118.775,249.366,-71.027,-178.503,9.925,149.564
C06903=1118.771,249.615,-71.056,-178.499,9.928,149.564
C06904=1118.766,249.863,-71.084,-178.495,9.932,149.564
C06905=1118.763,250.111,-71.112,-178.491,9.935,149.564
C06906=1118.758,250.360,-71.140,-178.487,9.938,149.563
C06907=1118.754,250.608,-71.169,-178.483,9.941,149.563
C06908=1118.750,250.856,-71.198,-178.480,9.943,149.563
C06909=1118.745,251.104,-71.226,-178.476,9.947,149.563
C06910=1118.741,251.353,-71.254,-178.473,9.949,149.562
C06911=1118.736,251.601,-71.282,-178.470,9.952,149.562
C06912=1118.732,251.849,-71.312,-178.467,9.955,149.562
C06913=1118.728,252.098,-71.340,-178.464,9.957,149.562
C06914=1118.723,252.346,-71.368,-178.460,9.960,149.561
C06915=1118.720,252.595,-71.396,-178.457,9.962,149.561
C06916=1118.716,252.808,-71.421,-178.456,9.964,149.561
C06917=1118.712,253.021,-71.446,-178.453,9.966,149.561
C06918=1118.709,253.234,-71.470,-178.452,9.968,149.561
C06919=1118.705,253.447,-71.495,-178.449,9.970,149.561
C06920=1118.702,253.660,-71.519,-178.448,9.971,149.561
C06921=1118.697,253.874,-71.544,-178.446,9.973,149.561
C06922=1118.694,254.087,-71.569,-178.444,9.975,149.561
C06923=1118.690,254.299,-71.593,-178.443,9.976,149.561
C06924=1118.686,254.548,-71.622,-178.441,9.979,149.561
C06925=1118.681,254.797,-71.650,-178.440,9.980,149.561
C06926=1118.677,255.044,-71.679,-178.438,9.982,149.561
C06927=1118.673,255.293,-71.708,-178.437,9.983,149.561
C06928=1118.669,255.542,-71.736,-178.436,9.985,149.561
C06929=1118.664,255.790,-71.765,-178.435,9.987,149.561
C06930=1118.660,256.038,-71.794,-178.434,9.989,149.562
C06931=1118.656,256.286,-71.823,-178.431,9.991,149.561
C06932=1118.652,256.535,-71.851,-178.428,9.994,149.561
C06933=1118.647,256.783,-71.880,-178.425,9.997,149.561
C06934=1118.643,257.031,-71.908,-178.423,10.000,149.561
C06935=1118.639,257.280,-71.937,-178.420,10.003,149.561
C06936=1118.634,257.528,-71.966,-178.417,10.006,149.561
C06937=1118.630,257.776,-71.994,-178.414,10.008,149.561
C06938=1118.626,258.025,-72.024,-178.411,10.011,149.561
C06939=1118.622,258.274,-72.053,-178.408,10.014,149.561
C06940=1118.618,258.521,-72.081,-178.405,10.017,149.561
C06941=1118.613,258.770,-72.110,-178.403,10.020,149.561
C06942=1118.609,259.018,-72.139,-178.400,10.022,149.561
C06943=1118.604,259.267,-72.168,-178.397,10.025,149.561
C06944=1118.600,259.514,-72.197,-178.394,10.028,149.560
C06945=1118.596,259.762,-72.226,-178.390,10.031,149.560
C06946=1118.592,260.011,-72.255,-178.387,10.034,149.560
C06947=1118.588,260.260,-72.284,-178.384,10.037,149.560
C06948=1118.584,260.508,-72.313,-178.381,10.040,149.560
C06949=1118.579,260.756,-72.341,-178.378,10.042,149.560
C06950=1118.575,261.004,-72.371,-178.375,10.045,149.560
C06951=1118.571,261.252,-72.400,-178.371,10.048,149.559
C06952=1118.566,261.501,-72.429,-178.368,10.051,149.559
C06953=1118.563,261.749,-72.458,-178.366,10.054,149.559
C06954=1118.558,261.997,-72.487,-178.363,10.057,149.559
C06955=1118.553,262.246,-72.516,-178.359,10.060,149.559
C06956=1118.549,262.494,-72.545,-178.356,10.063,149.559
C06957=1118.545,262.742,-72.575,-178.353,10.065,149.559
C06958=1118.541,262.990,-72.604,-178.349,10.069,149.559
C06959=1118.537,263.239,-72.634,-178.346,10.071,149.558
C06960=1118.532,263.488,-72.662,-178.343,10.074,149.558
C06961=1118.528,263.735,-72.691,-178.339,10.077,149.558
C06962=1118.524,263.983,-72.720,-178.336,10.080,149.558
C06963=1118.520,264.231,-72.750,-178.333,10.082,149.558
C06964=1118.516,264.480,-72.779,-178.329,10.086,149.557
C06965=1118.511,264.728,-72.809,-178.327,10.088,149.557
C06966=1118.507,264.976,-72.838,-178.324,10.091,149.557
C06967=1118.503,265.224,-72.868,-178.321,10.093,149.557
C06968=1118.499,265.473,-72.896,-178.319,10.095,149.557
C06969=1118.494,265.721,-72.925,-178.316,10.097,149.557
C06970=1118.490,265.969,-72.955,-178.313,10.100,149.557
C06971=1118.485,266.217,-72.984,-178.310,10.103,149.557
C06972=1118.482,266.430,-73.010,-178.308,10.105,149.557
C06973=1118.479,266.644,-73.035,-178.306,10.107,149.556
C06974=1118.475,266.857,-73.061,-178.303,10.109,149.556
C06975=1118.471,267.070,-73.085,-178.302,10.111,149.556
C06976=1118.468,267.282,-73.111,-178.299,10.113,149.556
C06977=1118.464,267.496,-73.136,-178.297,10.115,149.556
C06978=1118.461,267.709,-73.162,-178.294,10.118,149.556
C06979=1118.456,267.922,-73.186,-178.292,10.120,149.556
C06980=1118.453,268.170,-73.217,-178.289,10.122,149.556
C06981=1118.448,268.418,-73.246,-178.286,10.125,149.556
C06982=1118.444,268.666,-73.275,-178.283,10.127,149.556
C06983=1118.439,268.915,-73.306,-178.281,10.129,149.555
C06984=1118.435,269.163,-73.335,-178.278,10.132,149.555
C06985=1118.431,269.411,-73.364,-178.275,10.135,149.555
C06986=1118.427,269.660,-73.394,-178.272,10.138,149.555
C06987=1118.423,269.908,-73.423,-178.270,10.140,149.555
C06988=1118.419,270.156,-73.454,-178.267,10.142,149.555
C06989=1118.414,270.404,-73.483,-178.264,10.145,149.555
C06990=1118.410,270.652,-73.512,-178.261,10.148,149.555
C06991=1118.406,270.900,-73.542,-178.258,10.151,149.555
C06992=1118.401,271.149,-73.572,-178.256,10.153,149.554
C06993=1118.397,271.397,-73.602,-178.253,10.155,149.554
C06994=1118.393,271.645,-73.632,-178.250,10.158,149.554
C06995=1118.389,271.893,-73.661,-178.247,10.161,149.554
C06996=1118.385,272.141,-73.690,-178.244,10.164,149.554
C06997=1118.380,272.389,-73.721,-178.241,10.166,149.554
C06998=1118.376,272.638,-73.751,-178.238,10.169,149.554
C06999=1118.372,272.887,-73.780,-178.236,10.171,149.554
C07000=1118.368,273.134,-73.811,-178.233,10.174,149.554
C07001=1118.364,273.382,-73.840,-178.230,10.176,149.553
C07002=1118.359,273.631,-73.870,-178.227,10.179,149.553
C07003=1118.356,273.879,-73.900,-178.224,10.182,149.553
C07004=1118.351,274.127,-73.930,-178.221,10.185,149.553
C07005=1118.347,274.375,-73.960,-178.218,10.187,149.553
C07006=1118.343,274.623,-73.990,-178.215,10.190,149.553
C07007=1118.338,274.871,-74.019,-178.212,10.193,149.553
C07008=1118.334,275.119,-74.050,-178.209,10.195,149.552
C07009=1118.330,275.368,-74.080,-178.206,10.198,149.552
C07010=1118.326,275.616,-74.110,-178.203,10.201,149.552
C07011=1118.322,275.864,-74.140,-178.200,10.204,149.552
C07012=1118.318,276.112,-74.170,-178.197,10.206,149.552
C07013=1118.313,276.361,-74.200,-178.194,10.209,149.552
C07014=1118.309,276.608,-74.230,-178.191,10.212,149.552
C07015=1118.305,276.856,-74.259,-178.188,10.214,149.552
C07016=1118.301,277.104,-74.290,-178.185,10.217,149.551
C07017=1118.297,277.353,-74.321,-178.182,10.220,149.551
C07018=1118.292,277.601,-74.351,-178.179,10.222,149.551
C07019=1118.289,277.849,-74.381,-178.176,10.225,149.551
C07020=1118.284,278.097,-74.410,-178.172,10.227,149.551
C07021=1118.280,278.345,-74.441,-178.169,10.230,149.551
C07022=1118.277,278.594,-74.472,-178.166,10.233,149.550
C07023=1118.272,278.842,-74.502,-178.163,10.235,149.550
C07024=1118.268,279.090,-74.532,-178.160,10.238,149.550
C07025=1118.264,279.337,-74.562,-178.157,10.241,149.550
C07026=1118.259,279.586,-74.592,-178.154,10.243,149.550
C07027=1118.256,279.834,-74.623,-178.150,10.247,149.550
C07028=1118.252,280.047,-74.649,-178.148,10.249,149.549
C07029=1118.248,280.260,-74.675,-178.145,10.251,149.549
C07030=1118.244,280.473,-74.701,-178.142,10.253,149.549
C07031=1118.241,280.685,-74.727,-178.139,10.256,149.549
C07032=1118.237,280.898,-74.753,-178.137,10.258,149.549
C07033=1118.233,281.111,-74.780,-178.134,10.260,149.549
C07034=1118.230,281.324,-74.805,-178.131,10.262,149.548
C07035=1118.226,281.537,-74.832,-178.128,10.265,149.548
C07036=1118.222,281.786,-74.862,-178.125,10.267,149.548
C07037=1118.218,282.034,-74.892,-178.122,10.270,149.548
C07038=1118.214,282.282,-74.923,-178.119,10.273,149.548
C07039=1118.209,282.530,-74.953,-178.116,10.274,149.548
C07040=1118.205,282.778,-74.985,-178.113,10.277,149.547
C07041=1118.201,283.026,-75.015,-178.110,10.280,149.547
C07042=1118.197,283.274,-75.045,-178.107,10.282,149.547
C07043=1118.193,283.522,-75.076,-178.104,10.285,149.547
C07044=1118.189,283.770,-75.107,-178.101,10.288,149.547
C07045=1118.184,284.018,-75.138,-178.098,10.290,149.547
C07046=1118.180,284.266,-75.168,-178.094,10.293,149.546
C07047=1118.176,284.515,-75.198,-178.092,10.295,149.546
C07048=1118.172,284.763,-75.228,-178.089,10.297,149.546
C07049=1118.168,285.011,-75.259,-178.086,10.300,149.546
C07050=1118.164,285.259,-75.291,-178.083,10.303,149.546
C07051=1118.160,285.506,-75.321,-178.080,10.305,149.545
C07052=1118.155,285.754,-75.352,-178.077,10.308,149.545
C07053=1118.151,286.003,-75.383,-178.073,10.310,149.545
C07054=1118.147,286.251,-75.414,-178.070,10.313,149.545
C07055=1118.143,286.499,-75.444,-178.067,10.315,149.545
C07056=1118.139,286.747,-75.475,-178.064,10.318,149.545
C07057=1118.134,286.995,-75.506,-178.062,10.320,149.545
C07058=1118.131,287.244,-75.536,-178.058,10.323,149.544
C07059=1118.126,287.492,-75.567,-178.056,10.325,149.544
C07060=1118.122,287.739,-75.599,-178.052,10.328,149.544
C07061=1118.118,287.988,-75.630,-178.049,10.331,149.544
C07062=1118.114,288.235,-75.660,-178.046,10.333,149.543
C07063=1118.110,288.484,-75.691,-178.043,10.336,149.543
C07064=1118.106,288.732,-75.722,-178.040,10.338,149.543
C07065=1118.101,288.979,-75.753,-178.037,10.341,149.543
C07066=1118.097,289.228,-75.784,-178.034,10.344,149.543
C07067=1118.093,289.476,-75.815,-178.031,10.345,149.543
C07068=1118.089,289.724,-75.846,-178.028,10.348,149.543
C07069=1118.085,289.972,-75.877,-178.025,10.351,149.542
C07070=1118.081,290.220,-75.908,-178.022,10.353,149.542
C07071=1118.076,290.468,-75.939,-178.019,10.356,149.542
C07072=1118.072,290.715,-75.971,-178.016,10.358,149.542
C07073=1118.069,290.964,-76.001,-178.012,10.361,149.542
C07074=1118.064,291.212,-76.032,-178.009,10.364,149.541
C07075=1118.061,291.460,-76.064,-178.006,10.366,149.541
C07076=1118.056,291.708,-76.094,-178.004,10.368,149.541
C07077=1118.052,291.956,-76.126,-178.001,10.371,149.541
C07078=1118.048,292.204,-76.157,-177.997,10.373,149.541
C07079=1118.044,292.452,-76.188,-177.994,10.376,149.541
C07080=1118.039,292.700,-76.220,-177.991,10.378,149.540
C07081=1118.035,292.948,-76.251,-177.988,10.381,149.540
C07082=1118.032,293.195,-76.282,-177.985,10.384,149.540
C07083=1118.028,293.444,-76.313,-177.982,10.386,149.540
C07084=1118.024,293.657,-76.340,-177.980,10.388,149.540
C07085=1118.020,293.870,-76.367,-177.977,10.390,149.540
C07086=1118.016,294.082,-76.394,-177.974,10.393,149.539
C07087=1118.013,294.295,-76.421,-177.972,10.395,149.539
C07088=1118.010,294.508,-76.447,-177.969,10.397,149.539
C07089=1118.006,294.721,-76.474,-177.966,10.399,149.539
C07090=1118.002,294.934,-76.501,-177.964,10.401,149.539
C07091=1117.999,295.147,-76.528,-177.961,10.404,149.539
C07092=1117.995,295.394,-76.560,-177.958,10.406,149.538
C07093=1117.991,295.643,-76.591,-177.955,10.408,149.538
C07094=1117.987,295.890,-76.623,-177.952,10.411,149.538
C07095=1117.983,296.138,-76.654,-177.949,10.414,149.538
C07096=1117.978,296.386,-76.685,-177.946,10.416,149.538
C07097=1117.975,296.634,-76.717,-177.943,10.419,149.538
C07098=1117.970,296.882,-76.748,-177.939,10.421,149.537
C07099=1117.966,297.130,-76.780,-177.936,10.424,149.537
C07100=1117.963,297.378,-76.811,-177.933,10.426,149.537
C07101=1117.958,297.626,-76.843,-177.930,10.429,149.537
C07102=1117.954,297.874,-76.874,-177.927,10.431,149.537
C07103=1117.949,298.122,-76.906,-177.924,10.434,149.537
C07104=1117.946,298.370,-76.938,-177.921,10.436,149.536
C07105=1117.942,298.618,-76.970,-177.918,10.439,149.536
C07106=1117.937,298.865,-77.001,-177.915,10.441,149.536
C07107=1117.933,299.114,-77.032,-177.912,10.444,149.536
C07108=1117.930,299.362,-77.064,-177.909,10.446,149.536
C07109=1117.925,299.609,-77.096,-177.906,10.449,149.536
C07110=1117.921,299.858,-77.128,-177.902,10.452,149.535
C07111=1117.917,300.106,-77.160,-177.899,10.454,149.535
C07112=1117.913,300.353,-77.192,-177.897,10.456,149.535
C07113=1117.909,300.602,-77.223,-177.894,10.459,149.535
C07114=1117.905,300.850,-77.255,-177.890,10.461,149.535
C07115=1117.900,301.098,-77.287,-177.888,10.464,149.534
C07116=1117.897,301.346,-77.318,-177.884,10.466,149.534
C07117=1117.893,301.594,-77.350,-177.881,10.469,149.534
C07118=1117.889,301.841,-77.382,-177.878,10.472,149.534
C07119=1117.884,302.089,-77.414,-177.875,10.474,149.534
C07120=1117.880,302.337,-77.446,-177.872,10.477,149.533
C07121=1117.876,302.585,-77.478,-177.869,10.480,149.533
C07122=1117.872,302.833,-77.510,-177.865,10.482,149.533
C07123=1117.868,303.081,-77.542,-177.863,10.484,149.533
C07124=1117.864,303.328,-77.573,-177.860,10.486,149.533
C07125=1117.859,303.577,-77.606,-177.857,10.489,149.533
C07126=1117.855,303.825,-77.638,-177.853,10.492,149.532
C07127=1117.852,304.073,-77.669,-177.851,10.494,149.532
C07128=1117.847,304.320,-77.701,-177.847,10.497,149.532
C07129=1117.843,304.569,-77.733,-177.844,10.500,149.532
C07130=1117.840,304.816,-77.766,-177.841,10.502,149.532
C07131=1117.835,305.064,-77.798,-177.838,10.505,149.532
C07132=1117.831,305.312,-77.830,-177.835,10.507,149.531
C07133=1117.826,305.560,-77.862,-177.832,10.509,149.531
C07134=1117.823,305.808,-77.894,-177.829,10.512,149.531
C07135=1117.819,306.056,-77.926,-177.826,10.514,149.531
C07136=1117.814,306.303,-77.959,-177.823,10.517,149.531
C07137=1117.811,306.551,-77.991,-177.819,10.519,149.530
C07138=1117.806,306.799,-78.023,-177.817,10.522,149.530
C07139=1117.802,307.048,-78.055,-177.813,10.525,149.530
C07140=1117.799,307.259,-78.083,-177.811,10.527,149.530
C07141=1117.796,307.473,-78.110,-177.808,10.529,149.530
C07142=1117.791,307.685,-78.138,-177.805,10.531,149.530
C07143=1117.788,307.898,-78.165,-177.803,10.533,149.530
C07144=1117.785,308.110,-78.194,-177.800,10.536,149.529
C07145=1117.781,308.323,-78.221,-177.797,10.537,149.529
C07146=1117.778,308.536,-78.248,-177.795,10.539,149.529
C07147=1117.774,308.748,-78.277,-177.792,10.542,149.529
C07148=1117.770,308.996,-78.309,-177.789,10.545,149.529
C07149=1117.766,309.245,-78.341,-177.786,10.547,149.529
C07150=1117.763,309.492,-78.374,-177.783,10.549,149.528
C07151=1117.758,309.740,-78.406,-177.780,10.551,149.528
C07152=1117.754,309.987,-78.438,-177.777,10.554,149.528
C07153=1117.750,310.235,-78.471,-177.774,10.557,149.528
C07154=1117.746,310.483,-78.503,-177.771,10.559,149.528
C07155=1117.742,310.731,-78.536,-177.767,10.562,149.527
C07156=1117.738,310.979,-78.568,-177.764,10.565,149.527
C07157=1117.734,311.227,-78.601,-177.761,10.567,149.527
C07158=1117.730,311.475,-78.633,-177.758,10.570,149.527
C07159=1117.726,311.723,-78.666,-177.755,10.572,149.527
C07160=1117.722,311.971,-78.698,-177.751,10.575,149.527
C07161=1117.718,312.219,-78.731,-177.749,10.577,149.526
C07162=1117.714,312.466,-78.764,-177.746,10.579,149.526
C07163=1117.709,312.714,-78.796,-177.743,10.582,149.526
C07164=1117.706,312.961,-78.829,-177.740,10.584,149.526
C07165=1117.701,313.210,-78.861,-177.736,10.587,149.526
C07166=1117.697,313.457,-78.894,-177.733,10.590,149.526
C07167=1117.694,313.705,-78.927,-177.730,10.592,149.525
C07168=1117.689,313.953,-78.959,-177.727,10.595,149.525
C07169=1117.685,314.201,-78.992,-177.724,10.597,149.525
C07170=1117.682,314.448,-79.025,-177.721,10.600,149.525
C07171=1117.677,314.697,-79.057,-177.718,10.602,149.525
C07172=1117.673,314.944,-79.091,-177.714,10.605,149.524
C07173=1117.669,315.192,-79.124,-177.712,10.607,149.524
C07174=1117.665,315.440,-79.156,-177.709,10.609,149.524
C07175=1117.661,315.688,-79.189,-177.706,10.612,149.524
C07176=1117.657,315.936,-79.222,-177.702,10.615,149.524
C07177=1117.654,316.183,-79.254,-177.699,10.617,149.523
C07178=1117.649,316.431,-79.287,-177.696,10.620,149.523
C07179=1117.645,316.679,-79.320,-177.693,10.622,149.523
C07180=1117.641,316.927,-79.353,-177.690,10.625,149.523
C07181=1117.637,317.175,-79.386,-177.686,10.627,149.523
C07182=1117.633,317.422,-79.419,-177.683,10.630,149.523
C07183=1117.629,317.670,-79.452,-177.680,10.633,149.522
C07184=1117.625,317.918,-79.485,-177.677,10.635,149.522
C07185=1117.621,318.166,-79.518,-177.675,10.637,149.522
C07186=1117.617,318.414,-79.551,-177.671,10.639,149.522
C07187=1117.613,318.661,-79.583,-177.668,10.642,149.522
C07188=1117.609,318.909,-79.617,-177.665,10.645,149.522
C07189=1117.605,319.157,-79.650,-177.662,10.647,149.521
C07190=1117.601,319.405,-79.683,-177.658,10.650,149.521
C07191=1117.597,319.653,-79.716,-177.655,10.652,149.521
C07192=1117.593,319.900,-79.750,-177.652,10.655,149.521
C07193=1117.589,320.148,-79.783,-177.649,10.658,149.521
C07194=1117.586,320.395,-79.815,-177.646,10.660,149.520
C07195=1117.581,320.643,-79.848,-177.643,10.662,149.520
C07196=1117.578,320.856,-79.877,-177.640,10.664,149.520
C07197=1117.574,321.068,-79.905,-177.638,10.666,149.520
C07198=1117.571,321.281,-79.934,-177.635,10.669,149.520
C07199=1117.567,321.494,-79.963,-177.632,10.671,149.520
C07200=1117.564,321.706,-79.991,-177.630,10.673,149.519
C07201=1117.561,321.918,-80.020,-177.627,10.675,149.519
C07202=1117.558,322.131,-80.048,-177.624,10.677,149.519
C07203=1117.554,322.343,-80.077,-177.622,10.679,149.519
C07204=1117.549,322.591,-80.110,-177.618,10.681,149.519
C07205=1117.546,322.839,-80.143,-177.616,10.684,149.519
C07206=1117.542,323.087,-80.176,-177.612,10.687,149.518
C07207=1117.538,323.334,-80.210,-177.609,10.689,149.518
C07208=1117.534,323.582,-80.243,-177.606,10.692,149.518
C07209=1117.530,323.830,-80.277,-177.603,10.694,149.518
C07210=1117.526,324.078,-80.310,-177.600,10.697,149.518
C07211=1117.522,324.325,-80.344,-177.596,10.700,149.518
C07212=1117.518,324.573,-80.377,-177.593,10.702,149.517
C07213=1117.514,324.821,-80.410,-177.590,10.705,149.517
C07214=1117.510,325.068,-80.443,-177.587,10.707,149.517
C07215=1117.506,325.315,-80.477,-177.583,10.710,149.517
C07216=1117.503,325.564,-80.511,-177.581,10.712,149.517
C07217=1117.498,325.812,-80.544,-177.578,10.714,149.516
C07218=1117.495,326.059,-80.578,-177.575,10.717,149.516
C07219=1117.490,326.307,-80.612,-177.572,10.719,149.516
C07220=1117.486,326.555,-80.645,-177.568,10.722,149.516
C07221=1117.482,326.802,-80.679,-177.565,10.724,149.516
C07222=1117.478,327.050,-80.712,-177.562,10.727,149.516
C07223=1117.474,327.298,-80.745,-177.559,10.729,149.515
C07224=1117.471,327.546,-80.780,-177.555,10.732,149.515
C07225=1117.467,327.793,-80.813,-177.552,10.734,149.515
C07226=1117.462,328.041,-80.847,-177.549,10.737,149.515
C07227=1117.458,328.288,-80.880,-177.546,10.740,149.514
C07228=1117.455,328.536,-80.915,-177.543,10.741,149.514
C07229=1117.451,328.784,-80.948,-177.540,10.744,149.514
C07230=1117.447,329.031,-80.982,-177.537,10.747,149.514
C07231=1117.442,329.279,-81.015,-177.534,10.749,149.514
C07232=1117.439,329.527,-81.050,-177.531,10.752,149.514
C07233=1117.435,329.775,-81.083,-177.527,10.754,149.513
C07234=1117.431,330.022,-81.117,-177.524,10.757,149.513
C07235=1117.426,330.271,-81.151,-177.521,10.759,149.513
C07236=1117.423,330.518,-81.185,-177.518,10.762,149.513
C07237=1117.419,330.765,-81.219,-177.514,10.764,149.513
C07238=1117.415,331.013,-81.252,-177.511,10.767,149.512
C07239=1117.411,331.261,-81.286,-177.508,10.770,149.512
C07240=1117.407,331.508,-81.320,-177.506,10.771,149.512
C07241=1117.403,331.756,-81.354,-177.502,10.774,149.512
C07242=1117.399,332.004,-81.388,-177.499,10.776,149.512
C07243=1117.395,332.251,-81.422,-177.496,10.779,149.511
C07244=1117.391,332.499,-81.456,-177.493,10.781,149.511
C07245=1117.387,332.747,-81.490,-177.489,10.784,149.511
C07246=1117.383,332.994,-81.524,-177.486,10.787,149.511
C07247=1117.379,333.242,-81.558,-177.483,10.789,149.511
C07248=1117.375,333.489,-81.592,-177.480,10.791,149.510
C07249=1117.372,333.737,-81.626,-177.477,10.794,149.510
C07250=1117.367,333.985,-81.661,-177.474,10.797,149.510
C07251=1117.363,334.232,-81.695,-177.470,10.799,149.510
C07252=1117.360,334.445,-81.724,-177.468,10.801,149.510
C07253=1117.356,334.657,-81.753,-177.465,10.803,149.510
C07254=1117.353,334.869,-81.783,-177.462,10.806,149.510
C07255=1117.350,335.082,-81.812,-177.460,10.807,149.509
C07256=1117.347,335.294,-81.841,-177.457,10.809,149.509
C07257=1117.343,335.507,-81.871,-177.454,10.812,149.509
C07258=1117.339,335.719,-81.899,-177.452,10.814,149.509
C07259=1117.336,335.931,-81.929,-177.448,10.816,149.509
C07260=1117.333,336.179,-81.963,-177.446,10.818,149.508
C07261=1117.328,336.426,-81.998,-177.443,10.821,149.508
C07262=1117.325,336.674,-82.032,-177.440,10.823,149.508
C07263=1117.320,336.921,-82.066,-177.436,10.826,149.508
C07264=1117.317,337.169,-82.101,-177.433,10.828,149.508
C07265=1117.313,337.417,-82.135,-177.430,10.831,149.507
C07266=1117.309,337.664,-82.169,-177.427,10.833,149.507
C07267=1117.305,337.912,-82.204,-177.423,10.836,149.507
C07268=1117.301,338.159,-82.238,-177.420,10.838,149.507
C07269=1117.297,338.407,-82.272,-177.417,10.841,149.507
C07270=1117.293,338.654,-82.306,-177.414,10.843,149.507
C07271=1117.289,338.902,-82.341,-177.410,10.846,149.506
C07272=1117.285,339.150,-82.376,-177.408,10.848,149.506
C07273=1117.281,339.398,-82.410,-177.405,10.850,149.506
C07274=1117.277,339.645,-82.444,-177.402,10.853,149.506
C07275=1117.274,339.893,-82.479,-177.398,10.855,149.505
C07276=1117.269,340.140,-82.514,-177.395,10.858,149.505
C07277=1117.265,340.388,-82.549,-177.392,10.860,149.505
C07278=1117.262,340.635,-82.582,-177.389,10.863,149.505
C07279=1117.258,340.883,-82.617,-177.385,10.865,149.505
C07280=1117.253,341.130,-82.652,-177.382,10.868,149.504
C07281=1117.250,341.378,-82.686,-177.379,10.870,149.504
C07282=1117.245,341.625,-82.721,-177.375,10.873,149.504
C07283=1117.242,341.873,-82.756,-177.372,10.876,149.504
C07284=1117.238,342.121,-82.790,-177.369,10.878,149.504
C07285=1117.234,342.368,-82.825,-177.366,10.880,149.503
C07286=1117.230,342.616,-82.860,-177.363,10.882,149.503
C07287=1117.226,342.863,-82.894,-177.360,10.885,149.503
C07288=1117.222,343.111,-82.929,-177.357,10.887,149.503
C07289=1117.218,343.358,-82.964,-177.354,10.890,149.503
C07290=1117.214,343.606,-82.999,-177.350,10.892,149.503
C07291=1117.211,343.854,-83.033,-177.347,10.895,149.502
C07292=1117.207,344.101,-83.068,-177.344,10.897,149.502
C07293=1117.203,344.349,-83.103,-177.341,10.900,149.502
C07294=1117.198,344.596,-83.138,-177.337,10.902,149.502
C07295=1117.195,344.843,-83.173,-177.334,10.905,149.502
C07296=1117.191,345.091,-83.207,-177.331,10.907,149.501
C07297=1117.187,345.338,-83.243,-177.328,10.910,149.501
C07298=1117.183,345.586,-83.277,-177.325,10.912,149.501
C07299=1117.179,345.834,-83.313,-177.322,10.914,149.501
C07300=1117.175,346.081,-83.347,-177.319,10.917,149.501
C07301=1117.172,346.329,-83.382,-177.315,10.919,149.500
C07302=1117.168,346.577,-83.417,-177.312,10.922,149.500
C07303=1117.163,346.823,-83.452,-177.309,10.924,149.500
C07304=1117.159,347.072,-83.487,-177.305,10.927,149.500
C07305=1117.156,347.319,-83.523,-177.302,10.929,149.500
C07306=1117.152,347.566,-83.558,-177.299,10.932,149.499
C07307=1117.148,347.814,-83.593,-177.296,10.934,149.499
C07308=1117.144,348.026,-83.622,-177.293,10.936,149.499
C07309=1117.141,348.238,-83.653,-177.291,10.938,149.499
C07310=1117.138,348.450,-83.683,-177.288,10.940,149.499
C07311=1117.134,348.663,-83.713,-177.285,10.942,149.498
C07312=1117.131,348.874,-83.743,-177.282,10.945,149.498
C07313=1117.127,349.087,-83.773,-177.279,10.947,149.498
C07314=1117.125,349.299,-83.804,-177.277,10.949,149.498
C07315=1117.121,349.512,-83.834,-177.274,10.951,149.498
C07316=1117.117,349.759,-83.869,-177.270,10.954,149.497
C07317=1117.113,350.007,-83.904,-177.267,10.956,149.497
C07318=1117.110,350.254,-83.939,-177.264,10.958,149.497
C07319=1117.106,350.501,-83.974,-177.260,10.961,149.497
C07320=1117.102,350.748,-84.010,-177.257,10.963,149.497
